// TwinCAT 3 PLC project PowerLink_v2
// ProgramVersion: 3.1.4023.0
// libraries:
//   EfficientIO Communicator, * (EfficientIO)
//   EfficientIO ModbusTCP, * (EfficientIO)
//   Lynus Persistent Data V1, * (Lynus AG)
//   Lynus Standards, * (EfficientIO)
//   Tc2_BABasic, * (Beckhoff Automation GmbH)
//   Tc2_ModbusSrv, * (Beckhoff Automation GmbH)
//   Tc2_Standard, * (Beckhoff Automation GmbH)
//   Tc2_System, * (Beckhoff Automation GmbH)
//   Tc2_Utilities, * (Beckhoff Automation GmbH)
//   Tc3_IotBase, * (Beckhoff Automation GmbH)
//   Tc3_IPCDiag, * (Beckhoff Automation GmbH)
//   Tc3_JsonXml, * (Beckhoff Automation GmbH)
//   Tc3_Module, * (Beckhoff Automation GmbH)
//   EfficientIO Energy Basic,1.0.0.4,EfficientIO
// project tree:
//   DUTs/ ST_Hoymiles_DTU_Pro_PV_OutData.TcDUT (not stored)
//   ENUMs/ E_State.TcDUT
//   ENUMs/Hoymiles/ E_Hoymiles_OperatingState.TcDUT, E_Hoymiles_PV_Error.TcDUT
//   / FastTask.TcTTO (not stored), MiddleTask.TcTTO (not stored), SlowTask.TcTTO (not stored)
//   FBs/ FB_Convert_Dword_Real.TcPOU, FB_EM24_DIN.TcPOU (not stored), FB_Enphase.TcPOU (not stored), FB_ECS_LIBREO.TcPOU, FB_Enphase_Helper.TcPOU (not stored), FB_ECS_LIBREO_Helper.TcPOU, FB_Hoymiles_DTU_ProS_PV_Inverter.TcPOU, FB_Hoymiles_DTU_ProS_PV_Inverter_inclWrite.TcPOU, FB_ModBus_100Registers_FC3_inclID.TcPOU (not stored), FB_PAC2200.TcPOU, prg_ReadDeviceName.TcPOU
//   POUs/ prgBattery.TcPOU (not stored), prgCalc.TcPOU, prgComEffIO.TcPOU, prgCS.TcPOU, prgEM.TcPOU, prgEMS.TcPOU, prgEnphase.TcPOU (not stored), prgPersistent.TcPOU, prgPV.TcPOU, prgRWEffIO.TcPOU (not stored), prgSystemTime.TcPOU (not stored), prgVarEffIO.TcPOU (not stored)

// ---- ENUMs/E_State.TcDUT
{attribute 'qualified_only'}
TYPE E_State :
(
	Init := 0,
	ReadOnce,
	Error,
	Idle,
	Wait

	
);
END_TYPE

// ---- ENUMs/Hoymiles/E_Hoymiles_OperatingState.TcDUT
{attribute 'qualified_only'}
{attribute 'strict'}
TYPE E_Hoymiles_OperatingState :
(
	eNoDataReceived := 0,
	eOff := 1,
	eSleeping := 2,
	eStartingUp := 3,
	eTrackingPowerPoint := 4,
	eForcedPowerReduction := 5,
	eShuttingDown := 6,
	eFaults := 7,
	eStandby := 8
);
END_TYPE

// ---- ENUMs/Hoymiles/E_Hoymiles_PV_Error.TcDUT
{attribute 'qualified_only'}
{attribute 'strict'}
TYPE E_Hoymiles_PV_Error :
(
	eNoError := 0,
	eModbusTCPError := 1,
	eHoymilesError := 2,
	eHoymilesTooBigValueReceived := 3
);
END_TYPE

// ---- FBs/FB_Convert_Dword_Real.TcPOU
FUNCTION_BLOCK FB_Convert_Dword_Real
VAR_INPUT
	word_In_1:	WORD;
	word_In_2:	WORD;
	e_ByteOrderIn	: eByteOrder;						//Byte Format
	
END_VAR
VAR_OUTPUT
	real_Output	:REAL;
END_VAR
VAR
	fbConvertWordToDword		: FB_CV_WORD_TO_DWORD;			//Convert Word to Dword
	usintSign					: USINT;						// converstion dword to real	
	intExponent					: INT;							// converstion dword to real
	realMantisse				: REAL;							// converstion dword to real
END_VAR

fbConvertWordToDword(wInputValue_1:= word_In_1, wInputValue_2:= word_In_2, eByteOrderForConvert:= e_ByteOrderIn , dwOutputValue=> );
(* Sign *)
usintSign:=BOOL_TO_USINT(fbConvertWordToDword.dwOutputValue.31);
(* Exponent *)
intExponent:=DWORD_TO_INT(SHR(fbConvertWordToDword.dwOutputValue,23) AND 16#FF);
(* Mantisse *)
realMantisse:=DWORD_TO_REAL(fbConvertWordToDword.dwOutputValue AND 16#7FFFFF);
(* Result *)
real_Output := LREAL_TO_REAL((EXPT((-1),usintSign) * (1+realMantisse/8388608) * EXPT(2,intExponent-127)));

END_FUNCTION_BLOCK

// ---- FBs/FB_ECS_LIBREO.TcPOU
FUNCTION_BLOCK FB_ECS_LIBREO
VAR_INPUT
	bStart				: BOOL;
	tDelayRequest		: TIME := T#1S;		//Timer for delay before start with the next read or write Request
	sHostname			: STRING(255);		//Hostname or IP Adress from the Server
END_VAR

VAR_IN_OUT
END_VAR

VAR_OUTPUT
	bValidResult				: BOOL;															//Valid Result received from Server
    bBusy						: BOOL;															//Function is Busy
    bError						: BOOL;															//Error sucess
	bDone						: BOOL;															//True after the decoding from the received Json File
	bConnected					: BOOL;															//Connection to the Server
	hrErrorCode       			: HRESULT;														//Error Result from Http Client
	
	bCarConnected				: BOOL;
	bCarCharging				: BOOL;
	lrTotalPower				: LREAL;
	uiChrgCurr					: UINT;
	uiExtChrgCurr				: UINT;
END_VAR

VAR
	fbClient					: FB_IotHttpClient;
	fbHttpGet					: FB_ECS_LIBREO_Helper;
	timStartRequest				: TON;															//Timer to Start the Request
	FPStartRequest				: R_TRIG;														//Internal positive Edge
	FPDone						: R_TRIG;														//Internal positive Edge
	FNStart						: F_TRIG;														//Internal negative Edge
END_VAR

(*------------------------------------------------------------------------------------Configure HTTP Client------------------------------------------------------------------------------------------------------*)

fbClient.sHostName := sHostname;
fbClient.tConnectionTimeout := tDelayRequest;

IF NOT fbClient.bConfigured THEN 
	fbClient.nHostPort:= 80;
	fbClient.bKeepAlive := TRUE;
	fbClient.tConnectionTimeout := T#2S;
END_IF


//Timer to start the Request
FPStartRequest(CLK:= bStart, Q=> );
	timStartRequest(IN:= fbClient.bConfigured AND bStart AND NOT timStartRequest.Q, PT:= tDelayRequest, Q=> , ET=> );
		IF ((timStartRequest.Q AND NOT bBusy) OR (FPStartRequest.Q AND NOT bBusy AND fbClient.bConfigured)) THEN fbHttpGet.bSend := TRUE; END_IF

				
//Http Get Function
fbHttpGet(
	bCarConnected => bCarConnected, 
	bCarCharging => bCarCharging,
	lrTotalPower => lrTotalPower,
	uiChrgCurr => uiChrgCurr,
	uiExtChrgCurr => uiExtChrgCurr,
	bSend:= , 
	fbClient:= fbClient, 
	bBusy=> bBusy, 
	bError=> ,
	sContent=> );

lrTotalPower := LIMIT( 0, lrTotalPower, lrTotalPower) / 1000;

fbHttpGet.bSend := FALSE;

FPDone(CLK:= bDone, Q=> );

fbClient.Execute();

//Error
IF fbHttpGet.bError OR fbClient.bError THEN bError := TRUE; ELSE bError := FALSE; END_IF	
	hrErrorCode := fbClient.hrErrorCode;

END_FUNCTION_BLOCK

// ---- FBs/FB_ECS_LIBREO_Helper.TcPOU
FUNCTION_BLOCK FB_ECS_LIBREO_Helper
VAR_INPUT
	bSend			: BOOL;
END_VAR

VAR_IN_OUT
	fbClient		: FB_IotHttpClient;
END_VAR

VAR_OUTPUT
	bBusy					: BOOL;
	bError					: BOOL;
	bCarConnected			: BOOL;
	bCarCharging			: BOOL;
	lrTotalPower			: LREAL;
	uiChrgCurr				: UINT;
	uiExtChrgCurr			: UINT;

END_VAR

VAR
	fbRequestStatus		: FB_IotHttpRequest;
	fbJson				: FB_JsonDomParser;
	nState				: UDINT;
	RisingEdge			: R_TRIG;
	timTimeout			: TON;
	tTimeOut			: TIME := T#30S;
	
	bGetContentResult	: BOOL;
	sContent			: STRING(2048);
	
	bGetJsonResult		: BOOL;
	jsonDoc				: SJsonValue;
	jsonVal				: SJsonValue;
	
	nReqCount			: UDINT;	
	nResCount			: UDINT;
	nValidResCount		: UDINT;
	nErrCount			: UDINT;
END_VAR

//Timer for Timeout
timTimeout(IN:= nState = 1 AND bBusy, PT:= tTimeOut, Q=> , ET=> );
	IF timTimeout.Q THEN 
		nState := 0;
		bBusy := FALSE;
	END_IF

RisingEdge(CLK:= bSend );
CASE nState OF
0:	
	IF RisingEdge.Q THEN 
		IF fbRequestStatus.SendRequest(sUri:='/status', fbClient:=fbClient, eRequestType:=ETcIotHttpRequestType.HTTP_Get, 0, 0, 0) THEN
			nState:= 1;
			nReqCount:= nReqCount+1;
			bBusy:= TRUE;
			bError:= FALSE;
		END_IF					
	END_IF
1:
	IF NOT fbRequestStatus.bBusy THEN
		bError:= TRUE;
		
		IF NOT fbRequestStatus.bError THEN				 
			bGetContentResult:= fbRequestStatus.GetContent(pContent:= ADR(sContent), nContentSize:= SIZEOF(sContent), bSetNullTermination:= TRUE);
			IF fbRequestStatus.nStatusCode >= 200 AND fbRequestStatus.nStatusCode < 300 THEN
				bGetJsonResult:= FALSE;
				jsonDoc:= fbRequestStatus.GetJsonDomContent(fbJson);
				IF jsonDoc <> 0 THEN
					bGetJsonResult:= TRUE;
					IF fbJson.HasMember(jsonDoc, 'ts')  THEN
						jsonVal:= fbJson.FindMember(jsonDoc, 'chrgCurr');
						nValidResCount:= nValidResCount+1;
						IF fbJson.IsUint(jsonVal) THEN							
							uiChrgCurr:= UDINT_TO_UINT(fbJson.GetUint(jsonVal));									
						END_IF
						jsonVal:= fbJson.FindMember(jsonDoc, 'extCurr');
						nValidResCount:= nValidResCount+1;
						IF fbJson.IsUint(jsonVal) THEN							
							uiExtChrgCurr:= UDINT_TO_UINT(fbJson.GetUint(jsonVal));									
						END_IF
						jsonVal:= fbJson.FindMember(jsonDoc, 'evConn');
						nValidResCount:= nValidResCount+1;
						IF fbJson.IsBool(jsonVal) THEN							
							bCarConnected:= fbJson.GetBool(jsonVal);									
						END_IF
						jsonVal:= fbJson.FindMember(jsonDoc, 'chrgState');
						nValidResCount:= nValidResCount+1;
						IF fbJson.IsBool(jsonVal) THEN							
							bCarCharging:= fbJson.GetBool(jsonVal);									
						END_IF
						jsonVal:= fbJson.FindMemberPath(jsonDoc, 'readings/wattTotal');
						nValidResCount:= nValidResCount+1;
						IF fbJson.IsDouble(jsonVal) THEN							
							lrTotalPower:= fbJson.GetDouble(jsonVal);									
						END_IF		
						bError:= FALSE;
					END_IF						
				nResCount:= nResCount+1;			
				END_IF
			END_IF
		END_IF
		
	nState:= 0;
	bBusy:= FALSE;
		IF bError THEN
			nErrCount:= nErrCount+1;
		END_IF
	END_IF  	
END_CASE

fbClient.Execute();

END_FUNCTION_BLOCK

// ---- FBs/FB_Hoymiles_DTU_ProS_PV_Inverter.TcPOU
FUNCTION_BLOCK FB_Hoymiles_DTU_ProS_PV_Inverter
VAR_INPUT PERSISTENT
	bEnable						: BOOL;												//True = Function is enabled, FALSE = Function is dissabled, no new Data
	sIPAdress					: STRING(15);										//IP Adress from the Inverter
	byUnitID_Inverter			: BYTE;												//Unit ID fromt the Inverter (1 to 247)
END_VAR
VAR_OUTPUT
	DataHoymiles_DTU_Pro_Total	: ST_Hoymiles_DTU_Pro_PV_OutData;					//Output structure with Data from Symo 10
	arrDataHoymiles_DTU_Pro		: ARRAY[1..30] OF ST_Hoymiles_DTU_Pro_PV_OutData;	//Output structure with Data 
	stDataEMPower_PV			: ST_ElectricMeter_Output_Power;					//Output structure with Data from Electric Meter PV (Power Data)
	stDataEMCounter_PV			: ST_ElectricMeter_Output_Counter;					//Output structure with Data from Electric Meter PV (Counter Data)
	diNrOfEM_OUT_PV				: DINT;												//Active Number from the Electric Meter for using on other functions
END_VAR
VAR
	fbElMeter					: FB_ElectricMeter;									//Electric Meter Function 
	fbNumberDevice				: FB_NumberOfDevice;								//Function block to calcualte the number of the Device
	fbConvertEnergyRegister		: FB_CV_WORD_TO_UDINT;								//Convert function
	fbMBRead_FC3				: FB_MBReadRegs;									//Modbus Read Function (FC3)
	timDelay					: TON;												//Timer for Delay between Requests
	timTimeout					: TON;												//Timer for Timeout
	timDissableFunctions		: TON;												//Timer to dissable the Function after Lynus_Standards.Constants_General.tTimeDissableLynusFunctions Days without connection to the Lynus Cloud
	timResetConnectionOnGVL		: TON;												//Timer to try reset the connection Flag on the GVL. (When somebody delete the Connection Function and make only a onlinechange)
	FPEnable					: R_TRIG;											//Internal positive Edge
	FPError_FC_3				: R_TRIG;											//Internal positive Edge
	PD_String					: FB_PersistentData_String;							//Function to save persistent data 
	arrBuffer_FC3				: ARRAY[1..100] OF WORD;							//Buffer with Data from FC3
	arrPD						: ARRAY[1..2] OF FB_PersistentData_Number;			//Function to save persistent data 
	byWaitInStep				: BYTE;												//Wait in Step before start to clean data on PLC
	iStateGVLData				: INT;												//State machine to handle the data on the GVL
	iStateModbus				: INT;												//State variable for Statemachine
	iStateModbus_CP				: INT;												//Compare State variable
	diCounterForGVL				: DINT;												//Counter to clean old data on GVL
	rValBefWToOut				: REAL;												//Value to check the received data from the inverter befor wirte to the output structure
	lrCheckValue				: LREAL;											//Internal Value to check the value before convert
	i: INT;
	timDelayError: TON;
	x: INT;

	timWait: Ton;
END_VAR

//Creator : Stefan Lackner
//Company : EfficientIO
//Date : 02.05.2023
//Version : 0.0.0.0  NOT TESTED

//With this function its possible to read out values from the Hoymiles DTU ProS Gateway
//The protocol to the Inverter is Modbus TCP
//Attention. To access the registers, an offset of 1 must always be subtracted. Register 40001 would then be on register 40000.

// operation state of the inverter is unclear if that is ok, no documentation from Hoymiles

//NOTE for diNr.....Designation => 
//_IN = Here Data come in from other Functions or go out to other functions about the GVL
//_OUT = Here Data go out to other functions about the GVL

(*------------------------------------------------------------------------------------------General Input Part---------------------------------------------------------------------------------------------*)

//Check limitation
byUnitID_Inverter := LIMIT(1,byUnitID_Inverter,254);

(*-------------------------------------------------------------Calcualte the number of EM System---------------------------------------------------------------*)

fbNumberDevice(
	diActualNumberOfDevices:= Lynus_Standards.GVL_Energy.stNumberOfDevices.diNumberOfElectricMeters, 
	diMaxNumberOfDevices:= Constants_Energy.diMaxNumberOfElectricMeters, 
	udiCounterOnlineChange:= TwinCAT_SystemInfoVarList._AppInfo.OnlineChangeCnt, 
	bNumberIsCalculatet=> , 
	bFPNumberIsCalculatet=> , 
	bOnlineChange=> , 
	diNumberForThisDevice=> diNrOfEM_OUT_PV, 
	diNumberOfTotalDevices=> );

//Write new Numer on GVL
IF fbNumberDevice.bFPNumberIsCalculatet THEN
	Lynus_Standards.GVL_Energy.stNumberOfDevices.diNumberOfElectricMeters := fbNumberDevice.diNumberOfTotalDevices;	
END_IF 

//Delete old Number on GVL
IF fbNumberDevice.bOnlineChange THEN 
	Lynus_Standards.GVL_Energy.stNumberOfDevices.diNumberOfElectricMeters := diNrOfEM_OUT_PV;	
	iStateGVLData := 1; 
END_IF

(*-------------------------------------------------------------Service from Backend is ready and check the connection to backen for dissabel/enable Function---------------------------------------------------------------*)

//Try to reset the variable for connection on the GVL. When all is normal then the Lynus Mqtt connection function set this variable to true in the next cycle
//When we have no connection to the backend then after Lynus_Standards.Constants_General.tTimeDissableLynusFunctions days the Function is dissabled with all of his functionalities
timResetConnectionOnGVL(IN:= NOT timResetConnectionOnGVL.Q, PT:= T#1H, Q=> , ET=> );
IF timResetConnectionOnGVL.Q THEN Lynus_Standards.GVL_Communicator.bStateConnectionToEnableFunctions := FALSE; END_IF
IF NOT Lynus_Standards.GVL_Communicator.bStateConnectionToEnableFunctions THEN timDissableFunctions.IN := TRUE; ELSE timDissableFunctions.IN := FALSE; END_IF  
timDissableFunctions(IN:= , PT:= Lynus_Standards.Constants_General.tTimeDissableLynusFunctions, Q=> , ET=> );
	
(*------------------------------------------------------------------------------------------State Machine---------------------------------------------------------------------------------------------*)
	
//Enable
FPEnable(CLK:= bEnable, Q=> );
IF FPEnable.Q AND iStateModbus = 0 THEN iStateModbus := 1; END_IF
IF NOT bEnable OR timDissableFunctions.Q THEN iStateModbus := 0; END_IF

//Timer for delay
timDelay(IN:= , PT:= T#100MS, Q=> , ET=> );	

//Timer for Timeout in Statemachine
IF iStateModbus = iStateModbus_CP THEN timTimeout.IN := TRUE; ELSE timTimeout.IN := FALSE; END_IF
IF iStateModbus = 0 THEN timTimeout.IN := FALSE; END_IF
timTimeout(IN:= , PT:= T#20S, Q=> , ET=> );	

//Timer for delay in error state
timDelayError(IN:= , PT:= T#1S, Q=> , ET=> );	

// Timer for wait between polls
timWait(In:= , PT:= T#1S, Q=>, ET=> );


//Statemachine
CASE iStateModbus OF
	
	0://Init Step
		iStateModbus_CP := iStateModbus;
		timDelay.IN := FALSE;
		
		DataHoymiles_DTU_Pro_Total.bFunctionIsActive := FALSE;
		DataHoymiles_DTU_Pro_Total.eOperatingState := E_Hoymiles_OperatingState.eNoDataReceived;
		fbMBRead_FC3.bExecute := FALSE;
		lrCheckValue := 0;
		rValBefWToOut := 0;
		
		// clean arrays
		FOR i:=1 TO 30 BY 1 DO
			arrDataHoymiles_DTU_Pro[i].bError := FALSE;
			arrDataHoymiles_DTU_Pro[i].bFunctionIsActive := FALSE;
			arrDataHoymiles_DTU_Pro[i].eErrorState := 0;
			arrDataHoymiles_DTU_Pro[i].eOperatingState := 0;
			arrDataHoymiles_DTU_Pro[i].iPortNumber := 0;
			arrDataHoymiles_DTU_Pro[i].lrGridFrequency := 0;
			arrDataHoymiles_DTU_Pro[i].lrGridVoltage := 0;			
			arrDataHoymiles_DTU_Pro[i].lrPowerAcInverter := 0;
			arrDataHoymiles_DTU_Pro[i].lrPVVoltage := 0;
			arrDataHoymiles_DTU_Pro[i].lrPVCurrent := 0;
		END_FOR
		timDelayError.IN := TRUE;
		IF timDelayError.Q THEN
			iStateModbus := 1;
			timDelayError.IN := FALSE;
		END_IF				
			
	1://Read out first Registers from 4096 
		DataHoymiles_DTU_Pro_Total.bFunctionIsActive := TRUE;
		iStateModbus_CP := iStateModbus;
		
		fbMBRead_FC3.nQuantity := 100;
		fbMBRead_FC3.nMBAddr := 4096;
		fbMBRead_FC3.bExecute := TRUE;
		fbMBRead_FC3.nUnitID := byUnitID_Inverter;
			
		IF fbMBRead_FC3.bBusy THEN timDelay.IN := TRUE; END_IF
		
		//Wait for Delay, copy Data and then next step
		IF NOT fbMBRead_FC3.bBusy AND NOT fbMBRead_FC3.bError AND timDelay.Q THEN 
			FOR i:= 0 TO 4 BY 1 DO		// 5 ports per poll
				// Port Number
				arrDataHoymiles_DTU_Pro[i+1].iPortNumber := BYTE_TO_INT( WORD_TO_BYTE(arrBuffer_FC3[4+20*i] AND 16#FFFF));
				IF arrDataHoymiles_DTU_Pro[i+1].iPortNumber  <>0 THEN
					//PV Voltage
					arrDataHoymiles_DTU_Pro[i+1].lrPVVoltage  := (WORD_TO_LREAL(arrBuffer_FC3[5+20*i]))/10;
					//PV Current
					arrDataHoymiles_DTU_Pro[i+1].lrPVCurrent := (WORD_TO_LREAL(arrBuffer_FC3[6+20*i]))/100;
					//Grid Voltage
					arrDataHoymiles_DTU_Pro[i+1].lrGridVoltage := (WORD_TO_LREAL(arrBuffer_FC3[7+20*i]))/10;
					//Grid Frequency
					arrDataHoymiles_DTU_Pro[i+1].lrGridFrequency  := (WORD_TO_LREAL(arrBuffer_FC3[8+20*i]))/100;
					//Copy Data AC Power
					arrDataHoymiles_DTU_Pro[i+1].lrPowerAcInverter := (WORD_TO_LREAL(arrBuffer_FC3[9+20*i]))/10000;
				
					//Copy Data AC production Energy
			//		fbConvertEnergyRegister(wInputValue_1:= arrBuffer_FC3[11+20*i], wInputValue_2:= arrBuffer_FC3[12+20*i], eByteOrderForConvert:= eByteOrder.eBigEndian, udiOutputValue=> );
			//		rValBefWToOut := UDINT_TO_REAL(fbConvertEnergyRegister.udiOutputValue);
			//		lrCheckValue := rValBefWToOut;	
			//		IF lrCheckValue >= - 3.402823E+38 AND lrCheckValue <= 3.402823E+38 THEN 
			//			arrDataHoymiles_DTU_Pro[i+1].lrPVProductionEnergy := lrCheckValue /1000 ;
						arrDataHoymiles_DTU_Pro[i+1].lrPVProductionEnergy := (WORD_TO_REAL(arrBuffer_FC3[11+20*i]) * 65536 + WORD_TO_REAL(arrBuffer_FC3[12+20*i])) /10; 
			//		ELSE
			//			arrDataHoymiles_DTU_Pro[i+6].eErrorState := E_Hoymiles_PV_Error.eHoymilesTooBigValueReceived;	
			//		END_IF
					
					
					//Operating State		--->>>>> needs to get checked with Hoymiles if the states are correct
					IF arrBuffer_FC3[14+20*i] = 1 THEN 
						arrDataHoymiles_DTU_Pro[i+1].eOperatingState := E_Hoymiles_OperatingState.eOff;
					ELSIF arrBuffer_FC3[14+20*i] = 2 THEN 
						arrDataHoymiles_DTU_Pro[i+1].eOperatingState := E_Hoymiles_OperatingState.eSleeping;
					ELSIF arrBuffer_FC3[14+20*i] = 3 THEN 
						arrDataHoymiles_DTU_Pro[i+1].eOperatingState := E_Hoymiles_OperatingState.eStartingUp;
					ELSIF arrBuffer_FC3[14+20*i] = 4 THEN 
						arrDataHoymiles_DTU_Pro[i+1].eOperatingState := E_Hoymiles_OperatingState.eTrackingPowerPoint;
					ELSIF arrBuffer_FC3[14+20*i] = 5 THEN 
						arrDataHoymiles_DTU_Pro[i+1].eOperatingState := E_Hoymiles_OperatingState.eForcedPowerReduction;
					ELSIF arrBuffer_FC3[14+20*i] = 6 THEN 
						arrDataHoymiles_DTU_Pro[i+1].eOperatingState := E_Hoymiles_OperatingState.eShuttingDown;
					ELSIF arrBuffer_FC3[14+20*i] = 7 THEN 
						arrDataHoymiles_DTU_Pro[i+1].eOperatingState := E_Hoymiles_OperatingState.eFaults;
					ELSIF arrBuffer_FC3[14+20*i] = 8 THEN 
						arrDataHoymiles_DTU_Pro[i+1].eOperatingState := E_Hoymiles_OperatingState.eStandby;
					ELSE 
						arrDataHoymiles_DTU_Pro[i+1].eOperatingState := E_Hoymiles_OperatingState.eNoDataReceived;
					END_IF
				ELSE
					arrDataHoymiles_DTU_Pro[i+1].lrPVVoltage := 0;
					arrDataHoymiles_DTU_Pro[i+1].lrPVCurrent := 0;
					arrDataHoymiles_DTU_Pro[i+1].lrGridVoltage := 0;
					arrDataHoymiles_DTU_Pro[i+1].lrGridFrequency  := 0;
					arrDataHoymiles_DTU_Pro[i+1].lrPowerAcInverter := 0;
					arrDataHoymiles_DTU_Pro[i+1].lrPVProductionEnergy := 0;
				END_IF
			END_FOR
			//Next Step
			IF iStateModbus = 1 THEN
				fbMBRead_FC3.bExecute := FALSE;
				timDelay.IN := FALSE;
				iStateModbus := 2;
				DataHoymiles_DTU_Pro_Total.bError := FALSE; 
				DataHoymiles_DTU_Pro_Total.eErrorState := E_Hoymiles_PV_Error.eNoError;
			END_IF
		END_IF
			

		//Error or Timeout
		IF FPError_FC_3.Q OR timTimeout.Q THEN
			iStateModbus := 300;
			DataHoymiles_DTU_Pro_Total.eErrorState := E_Hoymiles_PV_Error.eModbusTCPError;
		END_IF

	2://Wait and back to 1 step or next ports poll
		iStateModbus_CP := iStateModbus;
		timWait.IN := TRUE;
		IF arrBuffer_FC3[82] <> 0 AND timWait.Q THEN // if the last port hast a serial number, so to the next 5 ports needs to get checked 
			timWait.IN := FALSE;
			iStateModbus := 3;
		ELSIF timWait.Q  THEN
			timWait.IN := FALSE;
			iStateModbus := 1;
		END_IF
	
	3://Read out second 100 Registers from 4296 
		DataHoymiles_DTU_Pro_Total.bFunctionIsActive := TRUE;
		iStateModbus_CP := iStateModbus;
		
		fbMBRead_FC3.nQuantity := 100;
		fbMBRead_FC3.nMBAddr := 4296;
		fbMBRead_FC3.bExecute := TRUE;
		fbMBRead_FC3.nUnitID := byUnitID_Inverter;
			
		IF fbMBRead_FC3.bBusy THEN timDelay.IN := TRUE; END_IF
		
		//Wait for Delay, copy Data and then next step
		IF NOT fbMBRead_FC3.bBusy AND NOT fbMBRead_FC3.bError AND timDelay.Q THEN 
			FOR i:= 0 TO 4 BY 1 DO		// 5 ports per poll
				// Port Number
				arrDataHoymiles_DTU_Pro[i+6].iPortNumber := BYTE_TO_INT( WORD_TO_BYTE(arrBuffer_FC3[4+20*i] AND 16#FFFF));
				IF arrDataHoymiles_DTU_Pro[i+6].iPortNumber <>0 THEN
					//PV Voltage
					arrDataHoymiles_DTU_Pro[i+6].lrPVVoltage  := (WORD_TO_LREAL(arrBuffer_FC3[5+20*i]))/10;
					//PV Current
					arrDataHoymiles_DTU_Pro[i+6].lrPVCurrent := (WORD_TO_LREAL(arrBuffer_FC3[6+20*i]))/100;
					//Grid Voltage
					arrDataHoymiles_DTU_Pro[i+6].lrGridVoltage := (WORD_TO_LREAL(arrBuffer_FC3[7+20*i]))/10;
					//Grid Frequency
					arrDataHoymiles_DTU_Pro[i+6].lrGridFrequency  := (WORD_TO_LREAL(arrBuffer_FC3[8+20*i]))/100;
					//Copy Data AC Power
					arrDataHoymiles_DTU_Pro[i+6].lrPowerAcInverter := (WORD_TO_LREAL(arrBuffer_FC3[9+20*i]))/10000;
				
					//Copy Data AC production Energy
			//		fbConvertEnergyRegister(wInputValue_1:= arrBuffer_FC3[11+20*i], wInputValue_2:= arrBuffer_FC3[12+20*i], eByteOrderForConvert:= eByteOrder.eBigEndian, udiOutputValue=> );
			//		rValBefWToOut := UDINT_TO_REAL(fbConvertEnergyRegister.udiOutputValue);
			//		lrCheckValue := rValBefWToOut;	
			//		IF lrCheckValue >= - 3.402823E+38 AND lrCheckValue <= 3.402823E+38 THEN 
			//			arrDataHoymiles_DTU_Pro[i+6].lrPVProductionEnergy := lrCheckValue /1000 ;
						arrDataHoymiles_DTU_Pro[i+6].lrPVProductionEnergy := (WORD_TO_REAL(arrBuffer_FC3[11+20*i]) * 65536 + WORD_TO_REAL(arrBuffer_FC3[12+20*i])) /10; 
			//		ELSE
			//			arrDataHoymiles_DTU_Pro[i+6].eErrorState := E_Hoymiles_PV_Error.eHoymilesTooBigValueReceived;	
			//		END_IF
					
					
					//Operating State		--->>>>> needs to get checked with Hoymiles if the states are correct
					IF arrBuffer_FC3[14+20*i] = 1 THEN 
						arrDataHoymiles_DTU_Pro[i+6].eOperatingState := E_Hoymiles_OperatingState.eOff;
					ELSIF arrBuffer_FC3[14+20*i] = 2 THEN 
						arrDataHoymiles_DTU_Pro[i+6].eOperatingState := E_Hoymiles_OperatingState.eSleeping;
					ELSIF arrBuffer_FC3[14+20*i] = 3 THEN 
						arrDataHoymiles_DTU_Pro[i+6].eOperatingState := E_Hoymiles_OperatingState.eStartingUp;
					ELSIF arrBuffer_FC3[14+20*i] = 4 THEN 
						arrDataHoymiles_DTU_Pro[i+6].eOperatingState := E_Hoymiles_OperatingState.eTrackingPowerPoint;
					ELSIF arrBuffer_FC3[14+20*i] = 5 THEN 
						arrDataHoymiles_DTU_Pro[i+6].eOperatingState := E_Hoymiles_OperatingState.eForcedPowerReduction;
					ELSIF arrBuffer_FC3[14+20*i] = 6 THEN 
						arrDataHoymiles_DTU_Pro[i+6].eOperatingState := E_Hoymiles_OperatingState.eShuttingDown;
					ELSIF arrBuffer_FC3[14+20*i] = 7 THEN 
						arrDataHoymiles_DTU_Pro[i+6].eOperatingState := E_Hoymiles_OperatingState.eFaults;
					ELSIF arrBuffer_FC3[14+20*i] = 8 THEN 
						arrDataHoymiles_DTU_Pro[i+6].eOperatingState := E_Hoymiles_OperatingState.eStandby;
					ELSE 
						arrDataHoymiles_DTU_Pro[i+6].eOperatingState := E_Hoymiles_OperatingState.eNoDataReceived;
					END_IF
				ELSE
					arrDataHoymiles_DTU_Pro[i+6].lrPVVoltage := 0;
					arrDataHoymiles_DTU_Pro[i+6].lrPVCurrent := 0;
					arrDataHoymiles_DTU_Pro[i+6].lrGridVoltage := 0;
					arrDataHoymiles_DTU_Pro[i+6].lrGridFrequency  := 0;
					arrDataHoymiles_DTU_Pro[i+6].lrPowerAcInverter := 0;
					arrDataHoymiles_DTU_Pro[i+6].lrPVProductionEnergy := 0;
				END_IF
			END_FOR
			//Next Step
			IF iStateModbus = 3 THEN
				fbMBRead_FC3.bExecute := FALSE;
				timDelay.IN := FALSE;
				iStateModbus := 4;
				DataHoymiles_DTU_Pro_Total.bError := FALSE; 
				DataHoymiles_DTU_Pro_Total.eErrorState := E_Hoymiles_PV_Error.eNoError;
			END_IF
		END_IF
		//Error or Timeout
		IF FPError_FC_3.Q OR timTimeout.Q THEN
			iStateModbus := 300;
			DataHoymiles_DTU_Pro_Total.eErrorState := E_Hoymiles_PV_Error.eModbusTCPError;
		END_IF
		
	4://Wait and back to 1 step
		iStateModbus_CP := iStateModbus;
		timWait.IN := TRUE;
		IF  arrBuffer_FC3[82] <> 0 AND timWait.Q THEN // if the last port hast a serial number, bo to the next 5 ports 
			timWait.IN := FALSE;
			iStateModbus := 1;		// change to state 5 and add the polls accordingly
		ELSIF timWait.Q  THEN
			timWait.IN := FALSE;
			iStateModbus := 1;
		END_IF
				
	300://Error
		iStateModbus_CP := iStateModbus;
		timDelay.IN := FALSE;
		fbMBRead_FC3.bExecute := FALSE;
		DataHoymiles_DTU_Pro_Total.bError := TRUE;
		timDelayError.IN := TRUE;
		IF timDelayError.Q THEN
			iStateModbus := 0;
			timDelayError.IN := FALSE;
		END_IF
							
END_CASE

(*------------------------------------------------------------------------------------------Modbus TCP Function---------------------------------------------------------------------------------------------*)

fbMBRead_FC3(	sIPAddr:= sIPAdress, 
				nTCPPort:= 502, 
				cbLength:= SIZEOF(arrBuffer_FC3), 
				pDestAddr:= ADR(arrBuffer_FC3), 
				tTimeout:= T#10S );
				
FPError_FC_3(CLK:= fbMBRead_FC3.bError, Q=> );

(*----------------------------------------------------------------------------------------Electric Meter Data----------------------------------------------------------------------------------------------*)

//Error and Warning
IF timDissableFunctions.Q THEN fbElMeter.bWarning := TRUE; fbElMeter.iWarningCode := 0; ELSE fbElMeter.bWarning := FALSE; END_IF   
IF DataHoymiles_DTU_Pro_Total.bError OR Lynus_Standards.GVL_Energy.stNumberOfDevices.diNumberOfElectricMeters > Constants_Energy.diMaxNumberOfElectricMeters THEN fbElMeter.bError := TRUE; ELSE fbElMeter.bError := FALSE; END_IF  

IF Lynus_Standards.GVL_Energy.stNumberOfDevices.diNumberOfElectricMeters > Constants_Energy.diMaxNumberOfElectricMeters THEN 
	fbElMeter.iErrorCode := 1;
ELSIF DataHoymiles_DTU_Pro_Total.bError THEN 
	fbElMeter.iErrorCode := 0;
END_IF  

//Read Out Data done for EM Function
IF iStateModbus <> 2 THEN fbElMeter.bReadOutDataDone := TRUE; ELSE fbElMeter.bReadOutDataDone := FALSE; END_IF

//Function block for meter data
IF iStateModbus = 2 OR iStateModbus = 4 THEN 
	fbElMeter.lrPowerTotal := 0;
	fbElMeter.lrFrequency := 0;
	FOR i:= 1 TO 30 BY 1 DO
		fbElMeter.lrPowerTotal := arrDataHoymiles_DTU_Pro[i].lrPowerAcInverter + fbElMeter.lrPowerTotal;
		IF arrDataHoymiles_DTU_Pro[i].lrGridFrequency > 45 AND arrDataHoymiles_DTU_Pro[i].lrGridFrequency < 55 THEN
			fbElMeter.lrFrequency := arrDataHoymiles_DTU_Pro[i].lrGridFrequency;
		END_IF
		IF arrDataHoymiles_DTU_Pro[i].lrGridVoltage >150 AND arrDataHoymiles_DTU_Pro[i].lrGridVoltage < 300 THEN
			fbElMeter.lrVoltageL1N := arrDataHoymiles_DTU_Pro[i].lrGridVoltage;
		END_IF
	END_FOR
END_IF
	
fbElMeter(
	bEnable:= bEnable AND NOT timDissableFunctions.Q, 
	bError:= , 
	bEnableReadOutFunction:= FALSE, 
	bWriteWithDelay:= TRUE,
	bPowerDataInvers:= TRUE, 
	bReadOutDataDone:= ,
	iTimeReadOutInterval:= , 
	iErrorCode:= , 
	iWarningCode:= , 
	lrTotalCounterEnergy_Consumption:= 0, 
	lrTotalCounterEnergy_Production:= , 
	lrCounterEnergyT1_Consumption:= 0, 
	lrCounterEnergyT2_Consumption:= 0, 
	lrCounterEnergyT1_Production:= , 
	lrCounterEnergyT2_Production:= 0, 
	lrCurrentL1:= 0, 
	lrVoltageL1N:= , 
	lrVoltageL1L2:= 0, 
	lrPowerL1:= 0, 
	lrCurrentL2:= 0, 
	lrVoltageL2N:= 0 , 
	lrVoltageL2L3:= 0 , 
	lrPowerL2:= 0, 
	lrCurrentL3:= 0 , 
	lrVoltageL3N:= 0, 
	lrVoltageL3L1:= 0, 
	lrPowerL3:= 0, 
	lrPowerTotal:= , 
	lrFrequency:= , 
	lrReactivePowerTotal:= 0, 
	lrApparentPowerTotal:= 0, 
	tTimDelayOutput:= T#5S, 
	stDataEMOutPower=> , 
	stDataEMOutPowerDelay=> stDataEMPower_PV, 
	stDataEMOutCounter=> ,
	stDataEMOutCounterDelay=> stDataEMCounter_PV, 
	bReadOutMeter=> );
DataHoymiles_DTU_Pro_Total.lrGridFrequency 		:= fbElMeter.lrFrequency;
DataHoymiles_DTU_Pro_Total.lrGridVoltage		:= fbElMeter.lrVoltageL1N;
DataHoymiles_DTU_Pro_Total.lrPowerAcInverter	:= fbElMeter.lrPowerTotal;
DataHoymiles_DTU_Pro_Total.lrPVProductionEnergy := stDataEMCounter_PV.lrTotalCounterEnergy_Production;

(*-----------------------------------------------------------Handle data to Global structure for the Electric Meter system-----------------------------------------------------------------*)

CASE iStateGVLData OF
	
	0://Init Step
		byWaitInStep := 0;
		diCounterForGVL := 1;
	
	1://Wait for 4 Steps before clean al Data on GVL
		byWaitInStep := byWaitInStep + 1;
		IF byWaitInStep >= 4 AND fbNumberDevice.bNumberIsCalculatet THEN iStateGVLData := 2; END_IF
		//To much Devices, back to the Init step
		IF byWaitInStep >= 4 AND NOT fbNumberDevice.bNumberIsCalculatet THEN iStateGVLData := 0; END_IF	
		
	2://Clear all Data in GVL
		Lynus_Standards.GVL_Energy.stDataElectricMeters[diCounterForGVL].bEnabled := FALSE;	
		Lynus_Standards.GVL_Energy.stDataElectricMeters[diCounterForGVL].byErrorWarning := 0;
		Lynus_Standards.GVL_Energy.stDataElectricMeters[diCounterForGVL].lrCounterEnergyT1_Consumption := 0;
		Lynus_Standards.GVL_Energy.stDataElectricMeters[diCounterForGVL].lrCounterEnergyT1_Production := 0;
		Lynus_Standards.GVL_Energy.stDataElectricMeters[diCounterForGVL].lrCounterEnergyT2_Consumption := 0;
		Lynus_Standards.GVL_Energy.stDataElectricMeters[diCounterForGVL].lrCounterEnergyT2_Production := 0;
		Lynus_Standards.GVL_Energy.stDataElectricMeters[diCounterForGVL].lrPower := 0;
		Lynus_Standards.GVL_Energy.stDataElectricMeters[diCounterForGVL].lrPowerConsumption := 0;
		Lynus_Standards.GVL_Energy.stDataElectricMeters[diCounterForGVL].lrPowerConsumption := 0;
		Lynus_Standards.GVL_Energy.stDataElectricMeters[diCounterForGVL].lrPowerProduction := 0;
		Lynus_Standards.GVL_Energy.stDataElectricMeters[diCounterForGVL].lrTotalCounterEnergy_Consumption := 0;
		Lynus_Standards.GVL_Energy.stDataElectricMeters[diCounterForGVL].lrTotalCounterEnergy_Production := 0;
		
		diCounterForGVL := diCounterForGVL + 1;
		diCounterForGVL := LIMIT(0,diCounterForGVL,Constants_Energy.diMaxNumberOfElectricMeters);
		//Back to the init step
		IF diCounterForGVL >= Constants_Energy.diMaxNumberOfElectricMeters THEN iStateGVLData := 0; END_IF
		
END_CASE 	 

IF diNrOfEM_OUT_PV > 0 AND fbNumberDevice.bNumberIsCalculatet THEN
	Lynus_Standards.GVL_Energy.stDataElectricMeters[diNrOfEM_OUT_PV].bEnabled := fbElMeter.stDataEMOutPower.bEnabled;
	Lynus_Standards.GVL_Energy.stDataElectricMeters[diNrOfEM_OUT_PV].byErrorWarning := fbElMeter.stDataEMOutPower.byErrorWarning;
	Lynus_Standards.GVL_Energy.stDataElectricMeters[diNrOfEM_OUT_PV].lrCounterEnergyT1_Consumption := fbElMeter.stDataEMOutCounter.lrCounterEnergyT1_Consumption;
	Lynus_Standards.GVL_Energy.stDataElectricMeters[diNrOfEM_OUT_PV].lrCounterEnergyT1_Production := fbElMeter.stDataEMOutCounter.lrCounterEnergyT1_Production;
	Lynus_Standards.GVL_Energy.stDataElectricMeters[diNrOfEM_OUT_PV].lrCounterEnergyT2_Consumption := fbElMeter.stDataEMOutCounter.lrCounterEnergyT2_Consumption;
	Lynus_Standards.GVL_Energy.stDataElectricMeters[diNrOfEM_OUT_PV].lrCounterEnergyT2_Production := fbElMeter.stDataEMOutCounter.lrCounterEnergyT2_Production;		
	Lynus_Standards.GVL_Energy.stDataElectricMeters[diNrOfEM_OUT_PV].lrPower := fbElMeter.stDataEMOutPower.lrPowerTotal;
	Lynus_Standards.GVL_Energy.stDataElectricMeters[diNrOfEM_OUT_PV].lrPowerConsumption := fbElMeter.stDataEMOutPower.lrPowerConsumption;
	Lynus_Standards.GVL_Energy.stDataElectricMeters[diNrOfEM_OUT_PV].lrPowerProduction := fbElMeter.stDataEMOutPower.lrPowerProduction;
	Lynus_Standards.GVL_Energy.stDataElectricMeters[diNrOfEM_OUT_PV].lrTotalCounterEnergy_Consumption := fbElMeter.stDataEMOutCounter.lrTotalCounterEnergy_Consumption;
	Lynus_Standards.GVL_Energy.stDataElectricMeters[diNrOfEM_OUT_PV].lrTotalCounterEnergy_Production := fbElMeter.stDataEMOutCounter.lrTotalCounterEnergy_Production;
END_IF

(*----------------------------------------------------------Save persistent data----------------------------------------------------------------*)

arrPD[1](lrValue:= BOOL_TO_LREAL(bEnable), bEventBasedActive=> );
arrPD[2](lrValue:= BYTE_TO_LREAL(byUnitID_Inverter), bEventBasedActive=> );
PD_String(sText:= sIPAdress, bEventBasedActive=> );

END_FUNCTION_BLOCK

// ---- FBs/FB_Hoymiles_DTU_ProS_PV_Inverter_inclWrite.TcPOU
FUNCTION_BLOCK FB_Hoymiles_DTU_ProS_PV_Inverter_inclWrite
VAR_INPUT PERSISTENT
	bEnable						: BOOL;												//True = Function is enabled, FALSE = Function is dissabled, no new Data
	sIPAdress					: STRING(15);										//IP Adress from the Inverter
	byUnitID_Inverter			: BYTE;												//Unit ID fromt the Inverter (1 to 247)
	byte_Setpoint				: BYTE;
END_VAR
VAR_OUTPUT
	DataHoymiles_DTU_Pro_Total	: ST_Hoymiles_DTU_Pro_PV_OutData;					//Output structure with Data from Symo 10
	arrDataHoymiles_DTU_Pro		: ARRAY[1..30] OF ST_Hoymiles_DTU_Pro_PV_OutData;	//Output structure with Data 
	stDataEMPower_PV			: ST_ElectricMeter_Output_Power;					//Output structure with Data from Electric Meter PV (Power Data)
	stDataEMCounter_PV			: ST_ElectricMeter_Output_Counter;					//Output structure with Data from Electric Meter PV (Counter Data)
	diNrOfEM_OUT_PV				: DINT;												//Active Number from the Electric Meter for using on other functions
END_VAR
VAR
	fbElMeter					: FB_ElectricMeter;									//Electric Meter Function 
	fbNumberDevice				: FB_NumberOfDevice;								//Function block to calcualte the number of the Device
	fbConvertEnergyRegister		: FB_CV_WORD_TO_UDINT;								//Convert function
	fbMBRead_FC3				: FB_MBReadRegs;									//Modbus Read Function (FC3)
	timDelay					: TON;												//Timer for Delay between Requests
	timTimeout					: TON;												//Timer for Timeout
	timDissableFunctions		: TON;												//Timer to dissable the Function after Lynus_Standards.Constants_General.tTimeDissableLynusFunctions Days without connection to the Lynus Cloud
	timResetConnectionOnGVL		: TON;												//Timer to try reset the connection Flag on the GVL. (When somebody delete the Connection Function and make only a onlinechange)
	FPEnable					: R_TRIG;											//Internal positive Edge
	FPError_FC_3				: R_TRIG;											//Internal positive Edge
	FPError_FC_6				: R_TRIG;											//Internal positive Edge
	PD_String					: FB_PersistentData_String;							//Function to save persistent data 
	arrBuffer_FC3				: ARRAY[1..100] OF WORD;							//Buffer with Data from FC3
	arrPD						: ARRAY[1..2] OF FB_PersistentData_Number;			//Function to save persistent data 
	byWaitInStep				: BYTE;												//Wait in Step before start to clean data on PLC
	iStateGVLData				: INT;												//State machine to handle the data on the GVL
	iStateModbus				: INT;												//State variable for Statemachine
	iStateModbus_CP				: INT;												//Compare State variable
	iStateModbusWrite			: INT;												//State variable for Statemachine
	diCounterForGVL				: DINT;												//Counter to clean old data on GVL
	rValBefWToOut				: REAL;												//Value to check the received data from the inverter befor wirte to the output structure
	lrCheckValue				: LREAL;											//Internal Value to check the value before convert
	i: INT;
	timDelayError: TON;
	x: INT;
	int_WriteSucessCounter: INT;
	fbMBWrite_FC6				: FB_MBWriteSingleReg;									//Modbus Write Function (FC16)
	timWait: Ton;
	
	wordBuffer_FC6				: WORD;								//Buffer with Data from FC6
	ton_Wait_write: Ton;
	tonDelayWrite: Ton;
	int_Error_Counter_Write: INT;
	ton_Wait_AfterWrite: TON;
END_VAR

//Creator : Stefan Lackner
//Company : EfficientIO
//Date : 02.05.2023
//Version : 0.0.0.0  NOT TESTED

//With this function its possible to read out values from the Hoymiles DTU ProS Gateway
//The protocol to the Inverter is Modbus TCP
//Attention. To access the registers, an offset of 1 must always be subtracted. Register 40001 would then be on register 40000.

// operation state of the inverter is unclear if that is ok, no documentation from Hoymiles

//NOTE for diNr.....Designation => 
//_IN = Here Data come in from other Functions or go out to other functions about the GVL
//_OUT = Here Data go out to other functions about the GVL

(*------------------------------------------------------------------------------------------General Input Part---------------------------------------------------------------------------------------------*)

//Check limitation
byUnitID_Inverter := LIMIT(1,byUnitID_Inverter,254);

(*-------------------------------------------------------------Calcualte the number of EM System---------------------------------------------------------------*)

fbNumberDevice(
	diActualNumberOfDevices:= Lynus_Standards.GVL_Energy.stNumberOfDevices.diNumberOfElectricMeters, 
	diMaxNumberOfDevices:= Constants_Energy.diMaxNumberOfElectricMeters, 
	udiCounterOnlineChange:= TwinCAT_SystemInfoVarList._AppInfo.OnlineChangeCnt, 
	bNumberIsCalculatet=> , 
	bFPNumberIsCalculatet=> , 
	bOnlineChange=> , 
	diNumberForThisDevice=> diNrOfEM_OUT_PV, 
	diNumberOfTotalDevices=> );

//Write new Numer on GVL
IF fbNumberDevice.bFPNumberIsCalculatet THEN
	Lynus_Standards.GVL_Energy.stNumberOfDevices.diNumberOfElectricMeters := fbNumberDevice.diNumberOfTotalDevices;	
END_IF 

//Delete old Number on GVL
IF fbNumberDevice.bOnlineChange THEN 
	Lynus_Standards.GVL_Energy.stNumberOfDevices.diNumberOfElectricMeters := diNrOfEM_OUT_PV;	
	iStateGVLData := 1; 
END_IF

(*-------------------------------------------------------------Service from Backend is ready and check the connection to backen for dissabel/enable Function---------------------------------------------------------------*)

//Try to reset the variable for connection on the GVL. When all is normal then the Lynus Mqtt connection function set this variable to true in the next cycle
//When we have no connection to the backend then after Lynus_Standards.Constants_General.tTimeDissableLynusFunctions days the Function is dissabled with all of his functionalities
timResetConnectionOnGVL(IN:= NOT timResetConnectionOnGVL.Q, PT:= T#1H, Q=> , ET=> );
IF timResetConnectionOnGVL.Q THEN Lynus_Standards.GVL_Communicator.bStateConnectionToEnableFunctions := FALSE; END_IF
IF NOT Lynus_Standards.GVL_Communicator.bStateConnectionToEnableFunctions THEN timDissableFunctions.IN := TRUE; ELSE timDissableFunctions.IN := FALSE; END_IF  
timDissableFunctions(IN:= , PT:= Lynus_Standards.Constants_General.tTimeDissableLynusFunctions, Q=> , ET=> );
	
(*------------------------------------------------------------------------------------------State Machine---------------------------------------------------------------------------------------------*)
	
//Enable
FPEnable(CLK:= bEnable, Q=> );
IF FPEnable.Q AND iStateModbus = 0 THEN iStateModbus := 1; END_IF
IF NOT bEnable OR timDissableFunctions.Q THEN iStateModbus := 0; END_IF

//Timer for delay
timDelay(IN:= , PT:= T#100MS, Q=> , ET=> );	
tonDelayWrite(IN:= , PT:= T#100MS, Q=> , ET=> );	

//Timer for Timeout in Statemachine
IF iStateModbus = iStateModbus_CP THEN timTimeout.IN := TRUE; ELSE timTimeout.IN := FALSE; END_IF
IF iStateModbus = 0 THEN timTimeout.IN := FALSE; END_IF
timTimeout(IN:= , PT:= T#20S, Q=> , ET=> );	

//Timer for delay in error state
timDelayError(IN:= , PT:= T#1S, Q=> , ET=> );	

// Timer for wait between polls
timWait(In:= , PT:= T#1S, Q=>, ET=> );


//Statemachine
CASE iStateModbus OF
	
	0://Init Step
		iStateModbus_CP := iStateModbus;
		timDelay.IN := FALSE;
		
		DataHoymiles_DTU_Pro_Total.bFunctionIsActive := FALSE;
		DataHoymiles_DTU_Pro_Total.eOperatingState := E_Hoymiles_OperatingState.eNoDataReceived;
		fbMBRead_FC3.bExecute := FALSE;
		lrCheckValue := 0;
		rValBefWToOut := 0;
		
		// clean arrays
		FOR i:=1 TO 30 BY 1 DO
			arrDataHoymiles_DTU_Pro[i].bError := FALSE;
			arrDataHoymiles_DTU_Pro[i].bFunctionIsActive := FALSE;
			arrDataHoymiles_DTU_Pro[i].eErrorState := 0;
			arrDataHoymiles_DTU_Pro[i].eOperatingState := 0;
			arrDataHoymiles_DTU_Pro[i].iPortNumber := 0;
			arrDataHoymiles_DTU_Pro[i].lrGridFrequency := 0;
			arrDataHoymiles_DTU_Pro[i].lrGridVoltage := 0;			
			arrDataHoymiles_DTU_Pro[i].lrPowerAcInverter := 0;
			arrDataHoymiles_DTU_Pro[i].lrPVVoltage := 0;
			arrDataHoymiles_DTU_Pro[i].lrPVCurrent := 0;
		END_FOR
		timDelayError.IN := TRUE;
		IF timDelayError.Q THEN
			iStateModbus := 1;
			timDelayError.IN := FALSE;
		END_IF				
			
	1://Read out first Registers from 4096 
		DataHoymiles_DTU_Pro_Total.bFunctionIsActive := TRUE;
		iStateModbus_CP := iStateModbus;
		
		fbMBRead_FC3.nQuantity := 100;
		fbMBRead_FC3.nMBAddr := 4096;
		fbMBRead_FC3.bExecute := TRUE;
		fbMBRead_FC3.nUnitID := byUnitID_Inverter;
			
		IF fbMBRead_FC3.bBusy THEN timDelay.IN := TRUE; END_IF
		
		//Wait for Delay, copy Data and then next step
		IF NOT fbMBRead_FC3.bBusy AND NOT fbMBRead_FC3.bError AND timDelay.Q THEN 
			FOR i:= 0 TO 4 BY 1 DO		// 5 ports per poll
				// Port Number
				arrDataHoymiles_DTU_Pro[i+1].iPortNumber := BYTE_TO_INT( WORD_TO_BYTE(arrBuffer_FC3[4+20*i] AND 16#FFFF));
				IF arrDataHoymiles_DTU_Pro[i+1].iPortNumber  <>0 THEN
					//PV Voltage
					arrDataHoymiles_DTU_Pro[i+1].lrPVVoltage  := (WORD_TO_LREAL(arrBuffer_FC3[5+20*i]))/10;
					//PV Current
					arrDataHoymiles_DTU_Pro[i+1].lrPVCurrent := (WORD_TO_LREAL(arrBuffer_FC3[6+20*i]))/100;
					//Grid Voltage
					arrDataHoymiles_DTU_Pro[i+1].lrGridVoltage := (WORD_TO_LREAL(arrBuffer_FC3[7+20*i]))/10;
					//Grid Frequency
					arrDataHoymiles_DTU_Pro[i+1].lrGridFrequency  := (WORD_TO_LREAL(arrBuffer_FC3[8+20*i]))/100;
					//Copy Data AC Power
					arrDataHoymiles_DTU_Pro[i+1].lrPowerAcInverter := (WORD_TO_LREAL(arrBuffer_FC3[9+20*i]))/10000;
				
					//Copy Data AC production Energy
			//		fbConvertEnergyRegister(wInputValue_1:= arrBuffer_FC3[11+20*i], wInputValue_2:= arrBuffer_FC3[12+20*i], eByteOrderForConvert:= eByteOrder.eBigEndian, udiOutputValue=> );
			//		rValBefWToOut := UDINT_TO_REAL(fbConvertEnergyRegister.udiOutputValue);
			//		lrCheckValue := rValBefWToOut;	
			//		IF lrCheckValue >= - 3.402823E+38 AND lrCheckValue <= 3.402823E+38 THEN 
			//			arrDataHoymiles_DTU_Pro[i+1].lrPVProductionEnergy := lrCheckValue /1000 ;
						arrDataHoymiles_DTU_Pro[i+1].lrPVProductionEnergy := (WORD_TO_REAL(arrBuffer_FC3[11+20*i]) * 65536 + WORD_TO_REAL(arrBuffer_FC3[12+20*i])) /10; 
			//		ELSE
			//			arrDataHoymiles_DTU_Pro[i+6].eErrorState := E_Hoymiles_PV_Error.eHoymilesTooBigValueReceived;	
			//		END_IF
					
					
					//Operating State		--->>>>> needs to get checked with Hoymiles if the states are correct
					IF arrBuffer_FC3[14+20*i] = 1 THEN 
						arrDataHoymiles_DTU_Pro[i+1].eOperatingState := E_Hoymiles_OperatingState.eOff;
					ELSIF arrBuffer_FC3[14+20*i] = 2 THEN 
						arrDataHoymiles_DTU_Pro[i+1].eOperatingState := E_Hoymiles_OperatingState.eSleeping;
					ELSIF arrBuffer_FC3[14+20*i] = 3 THEN 
						arrDataHoymiles_DTU_Pro[i+1].eOperatingState := E_Hoymiles_OperatingState.eStartingUp;
					ELSIF arrBuffer_FC3[14+20*i] = 4 THEN 
						arrDataHoymiles_DTU_Pro[i+1].eOperatingState := E_Hoymiles_OperatingState.eTrackingPowerPoint;
					ELSIF arrBuffer_FC3[14+20*i] = 5 THEN 
						arrDataHoymiles_DTU_Pro[i+1].eOperatingState := E_Hoymiles_OperatingState.eForcedPowerReduction;
					ELSIF arrBuffer_FC3[14+20*i] = 6 THEN 
						arrDataHoymiles_DTU_Pro[i+1].eOperatingState := E_Hoymiles_OperatingState.eShuttingDown;
					ELSIF arrBuffer_FC3[14+20*i] = 7 THEN 
						arrDataHoymiles_DTU_Pro[i+1].eOperatingState := E_Hoymiles_OperatingState.eFaults;
					ELSIF arrBuffer_FC3[14+20*i] = 8 THEN 
						arrDataHoymiles_DTU_Pro[i+1].eOperatingState := E_Hoymiles_OperatingState.eStandby;
					ELSE 
						arrDataHoymiles_DTU_Pro[i+1].eOperatingState := E_Hoymiles_OperatingState.eNoDataReceived;
					END_IF
				ELSE
					arrDataHoymiles_DTU_Pro[i+1].lrPVVoltage := 0;
					arrDataHoymiles_DTU_Pro[i+1].lrPVCurrent := 0;
					arrDataHoymiles_DTU_Pro[i+1].lrGridVoltage := 0;
					arrDataHoymiles_DTU_Pro[i+1].lrGridFrequency  := 0;
					arrDataHoymiles_DTU_Pro[i+1].lrPowerAcInverter := 0;
					arrDataHoymiles_DTU_Pro[i+1].lrPVProductionEnergy := 0;
				END_IF
			END_FOR
			//Next Step
			IF iStateModbus = 1 THEN
				fbMBRead_FC3.bExecute := FALSE;
				timDelay.IN := FALSE;
				iStateModbus := 2;
				DataHoymiles_DTU_Pro_Total.bError := FALSE; 
				DataHoymiles_DTU_Pro_Total.eErrorState := E_Hoymiles_PV_Error.eNoError;
			END_IF
		END_IF
			

		//Error or Timeout
		IF FPError_FC_3.Q OR timTimeout.Q THEN
			iStateModbus := 300;
			DataHoymiles_DTU_Pro_Total.eErrorState := E_Hoymiles_PV_Error.eModbusTCPError;
		END_IF

	2://Wait and back to 1 step or next ports poll
		iStateModbus_CP := iStateModbus;
		timWait.IN := TRUE;
		IF arrBuffer_FC3[82] <> 0 AND timWait.Q THEN // if the last port hast a serial number, so to the next 5 ports needs to get checked 
			timWait.IN := FALSE;
			iStateModbus := 3;
		ELSIF timWait.Q  THEN
			timWait.IN := FALSE;
			iStateModbusWrite := 1;
			iStateModbus := -1;
			iStateModbus_CP := iStateModbus;
			// iStateModbus := 1;
		END_IF
	
	3://Read out second 100 Registers from 4296 
		DataHoymiles_DTU_Pro_Total.bFunctionIsActive := TRUE;
		iStateModbus_CP := iStateModbus;
		
		fbMBRead_FC3.nQuantity := 100;
		fbMBRead_FC3.nMBAddr := 4296;
		fbMBRead_FC3.bExecute := TRUE;
		fbMBRead_FC3.nUnitID := byUnitID_Inverter;
			
		IF fbMBRead_FC3.bBusy THEN timDelay.IN := TRUE; END_IF
		
		//Wait for Delay, copy Data and then next step
		IF NOT fbMBRead_FC3.bBusy AND NOT fbMBRead_FC3.bError AND timDelay.Q THEN 
			FOR i:= 0 TO 4 BY 1 DO		// 5 ports per poll
				// Port Number
				arrDataHoymiles_DTU_Pro[i+6].iPortNumber := BYTE_TO_INT( WORD_TO_BYTE(arrBuffer_FC3[4+20*i] AND 16#FFFF));
				IF arrDataHoymiles_DTU_Pro[i+6].iPortNumber <>0 THEN
					//PV Voltage
					arrDataHoymiles_DTU_Pro[i+6].lrPVVoltage  := (WORD_TO_LREAL(arrBuffer_FC3[5+20*i]))/10;
					//PV Current
					arrDataHoymiles_DTU_Pro[i+6].lrPVCurrent := (WORD_TO_LREAL(arrBuffer_FC3[6+20*i]))/100;
					//Grid Voltage
					arrDataHoymiles_DTU_Pro[i+6].lrGridVoltage := (WORD_TO_LREAL(arrBuffer_FC3[7+20*i]))/10;
					//Grid Frequency
					arrDataHoymiles_DTU_Pro[i+6].lrGridFrequency  := (WORD_TO_LREAL(arrBuffer_FC3[8+20*i]))/100;
					//Copy Data AC Power
					arrDataHoymiles_DTU_Pro[i+6].lrPowerAcInverter := (WORD_TO_LREAL(arrBuffer_FC3[9+20*i]))/10000;
				
					//Copy Data AC production Energy
			//		fbConvertEnergyRegister(wInputValue_1:= arrBuffer_FC3[11+20*i], wInputValue_2:= arrBuffer_FC3[12+20*i], eByteOrderForConvert:= eByteOrder.eBigEndian, udiOutputValue=> );
			//		rValBefWToOut := UDINT_TO_REAL(fbConvertEnergyRegister.udiOutputValue);
			//		lrCheckValue := rValBefWToOut;	
			//		IF lrCheckValue >= - 3.402823E+38 AND lrCheckValue <= 3.402823E+38 THEN 
			//			arrDataHoymiles_DTU_Pro[i+6].lrPVProductionEnergy := lrCheckValue /1000 ;
						arrDataHoymiles_DTU_Pro[i+6].lrPVProductionEnergy := (WORD_TO_REAL(arrBuffer_FC3[11+20*i]) * 65536 + WORD_TO_REAL(arrBuffer_FC3[12+20*i])) /10; 
			//		ELSE
			//			arrDataHoymiles_DTU_Pro[i+6].eErrorState := E_Hoymiles_PV_Error.eHoymilesTooBigValueReceived;	
			//		END_IF
					
					
					//Operating State		--->>>>> needs to get checked with Hoymiles if the states are correct
					IF arrBuffer_FC3[14+20*i] = 1 THEN 
						arrDataHoymiles_DTU_Pro[i+6].eOperatingState := E_Hoymiles_OperatingState.eOff;
					ELSIF arrBuffer_FC3[14+20*i] = 2 THEN 
						arrDataHoymiles_DTU_Pro[i+6].eOperatingState := E_Hoymiles_OperatingState.eSleeping;
					ELSIF arrBuffer_FC3[14+20*i] = 3 THEN 
						arrDataHoymiles_DTU_Pro[i+6].eOperatingState := E_Hoymiles_OperatingState.eStartingUp;
					ELSIF arrBuffer_FC3[14+20*i] = 4 THEN 
						arrDataHoymiles_DTU_Pro[i+6].eOperatingState := E_Hoymiles_OperatingState.eTrackingPowerPoint;
					ELSIF arrBuffer_FC3[14+20*i] = 5 THEN 
						arrDataHoymiles_DTU_Pro[i+6].eOperatingState := E_Hoymiles_OperatingState.eForcedPowerReduction;
					ELSIF arrBuffer_FC3[14+20*i] = 6 THEN 
						arrDataHoymiles_DTU_Pro[i+6].eOperatingState := E_Hoymiles_OperatingState.eShuttingDown;
					ELSIF arrBuffer_FC3[14+20*i] = 7 THEN 
						arrDataHoymiles_DTU_Pro[i+6].eOperatingState := E_Hoymiles_OperatingState.eFaults;
					ELSIF arrBuffer_FC3[14+20*i] = 8 THEN 
						arrDataHoymiles_DTU_Pro[i+6].eOperatingState := E_Hoymiles_OperatingState.eStandby;
					ELSE 
						arrDataHoymiles_DTU_Pro[i+6].eOperatingState := E_Hoymiles_OperatingState.eNoDataReceived;
					END_IF
				ELSE
					arrDataHoymiles_DTU_Pro[i+6].lrPVVoltage := 0;
					arrDataHoymiles_DTU_Pro[i+6].lrPVCurrent := 0;
					arrDataHoymiles_DTU_Pro[i+6].lrGridVoltage := 0;
					arrDataHoymiles_DTU_Pro[i+6].lrGridFrequency  := 0;
					arrDataHoymiles_DTU_Pro[i+6].lrPowerAcInverter := 0;
					arrDataHoymiles_DTU_Pro[i+6].lrPVProductionEnergy := 0;
				END_IF
			END_FOR
			//Next Step
			IF iStateModbus = 3 THEN
				fbMBRead_FC3.bExecute := FALSE;
				timDelay.IN := FALSE;
				iStateModbus := 4;
				DataHoymiles_DTU_Pro_Total.bError := FALSE; 
				DataHoymiles_DTU_Pro_Total.eErrorState := E_Hoymiles_PV_Error.eNoError;
			END_IF
		END_IF
		//Error or Timeout
		IF FPError_FC_3.Q OR timTimeout.Q THEN
			iStateModbus := 300;
			DataHoymiles_DTU_Pro_Total.eErrorState := E_Hoymiles_PV_Error.eModbusTCPError;
		END_IF
		
	4://Wait and back to 1 step
		iStateModbus_CP := iStateModbus;
		timWait.IN := TRUE;
		IF  arrBuffer_FC3[82] <> 0 AND timWait.Q THEN // if the last port hast a serial number, bo to the next 5 ports 
			timWait.IN := FALSE;
			iStateModbus := 1;		// change to state 5 and add the polls accordingly
		ELSIF timWait.Q  THEN
			timWait.IN := FALSE;
			iStateModbus := -1;
			iStateModbusWrite := 1;
			iStateModbus_CP := iStateModbus;
		//	iStateModbus := 1;
		END_IF
				
	300://Error
		iStateModbus_CP := iStateModbus;
		timDelay.IN := FALSE;
		fbMBRead_FC3.bExecute := FALSE;
		DataHoymiles_DTU_Pro_Total.bError := TRUE;
		timDelayError.IN := TRUE;
		IF timDelayError.Q THEN
			iStateModbus := 0;
			timDelayError.IN := FALSE;
		END_IF
							
END_CASE

(*------------------------------------------------------------------------------------------WriteFunction---------------------------------------------------------------------------------------------*)

	
CASE iStateModbusWrite OF	
	1://Search the Unit ID to read out the Data for each Inverter with Unit ID <> 0
		//iStateModbus_CP := iStateModbusWrite;
		byte_Setpoint := LIMIT (0,byte_Setpoint,100);
		
		iStateModbusWrite := 2;
				

	2://write setpoint
		//iStateModbus_CP := iStateModbusWrite;	

		wordBuffer_FC6 := BYTE_TO_WORD(byte_Setpoint);


		fbMBWrite_FC6.nMBAddr := 16#C001;
		fbMBWrite_FC6.bExecute := TRUE;
		fbMBWrite_FC6.nValue:= wordBuffer_FC6; 

				
		IF fbMBWrite_FC6.bBusy THEN 
			tonDelayWrite.IN := TRUE; 
		END_IF
	
		//Wait for Delay and then next step
		IF NOT fbMBWrite_FC6.bBusy AND NOT fbMBWrite_FC6.bError AND tonDelayWrite.Q THEN

			int_WriteSucessCounter :=int_WriteSucessCounter+1;
			
			fbMBWrite_FC6.bExecute := FALSE;
			tonDelayWrite.IN := FALSE;
			//Restart from new with the Read out part
			iStateModbusWrite := 3;
		END_IF
				
		//Error or Timout
		IF FPError_FC_6.Q OR timTimeout.Q THEN
			fbMBWrite_FC6.bExecute := FALSE;
			tonDelayWrite.IN := FALSE;
			iStateModbusWrite := 300;
		END_IF
	
	3:
		ton_Wait_AfterWrite.IN:=TRUE;
		IF ton_Wait_AfterWrite.Q THEN
			ton_Wait_AfterWrite.IN:=FALSE;
			iStateModbus := 1;
			iStateModbusWrite := 0;
		END_IF
		
		
	300:   // error
		int_Error_Counter_Write := int_Error_Counter_Write+1;
		iStateModbus := 1;
		iStateModbusWrite := 0;
END_CASE
ton_Wait_AfterWrite(pt:= T#2S);


(*------------------------------------------------------------------------------------------Modbus TCP Function---------------------------------------------------------------------------------------------*)

fbMBRead_FC3(	sIPAddr:= sIPAdress, 
				nTCPPort:= 502, 
				cbLength:= SIZEOF(arrBuffer_FC3), 
				pDestAddr:= ADR(arrBuffer_FC3), 
				tTimeout:= T#10S );
				
FPError_FC_3(CLK:= fbMBRead_FC3.bError, Q=> );

fbMBWrite_FC6(
	sIPAddr:= sIPAdress , 
	nTCPPort:= 502, 
	nUnitID:= byUnitID_Inverter, 
	nMBAddr:= , 
	nValue:= , 
	bExecute:= , 
	tTimeout:= T#5S, 
	bBusy=> , 
	bError=> , 
	nErrId=> );


		
FPError_FC_6(CLK:= fbMBWrite_FC6.bError, Q=> );



(*----------------------------------------------------------------------------------------Electric Meter Data----------------------------------------------------------------------------------------------*)

//Error and Warning
IF timDissableFunctions.Q THEN fbElMeter.bWarning := TRUE; fbElMeter.iWarningCode := 0; ELSE fbElMeter.bWarning := FALSE; END_IF   
IF DataHoymiles_DTU_Pro_Total.bError OR Lynus_Standards.GVL_Energy.stNumberOfDevices.diNumberOfElectricMeters > Constants_Energy.diMaxNumberOfElectricMeters THEN fbElMeter.bError := TRUE; ELSE fbElMeter.bError := FALSE; END_IF  

IF Lynus_Standards.GVL_Energy.stNumberOfDevices.diNumberOfElectricMeters > Constants_Energy.diMaxNumberOfElectricMeters THEN 
	fbElMeter.iErrorCode := 1;
ELSIF DataHoymiles_DTU_Pro_Total.bError THEN 
	fbElMeter.iErrorCode := 0;
END_IF  

//Read Out Data done for EM Function
IF iStateModbus <> 2 THEN fbElMeter.bReadOutDataDone := TRUE; ELSE fbElMeter.bReadOutDataDone := FALSE; END_IF

//Function block for meter data
IF iStateModbus = 2 OR iStateModbus = 4 THEN 
	fbElMeter.lrPowerTotal := 0;
	fbElMeter.lrFrequency := 0;
	FOR i:= 1 TO 30 BY 1 DO
		fbElMeter.lrPowerTotal := arrDataHoymiles_DTU_Pro[i].lrPowerAcInverter + fbElMeter.lrPowerTotal;
		IF arrDataHoymiles_DTU_Pro[i].lrGridFrequency > 45 AND arrDataHoymiles_DTU_Pro[i].lrGridFrequency < 55 THEN
			fbElMeter.lrFrequency := arrDataHoymiles_DTU_Pro[i].lrGridFrequency;
		END_IF
		IF arrDataHoymiles_DTU_Pro[i].lrGridVoltage >150 AND arrDataHoymiles_DTU_Pro[i].lrGridVoltage < 300 THEN
			fbElMeter.lrVoltageL1N := arrDataHoymiles_DTU_Pro[i].lrGridVoltage;
		END_IF
	END_FOR
END_IF
	
fbElMeter(
	bEnable:= bEnable AND NOT timDissableFunctions.Q, 
	bError:= , 
	bEnableReadOutFunction:= FALSE, 
	bWriteWithDelay:= TRUE,
	bPowerDataInvers:= TRUE, 
	bReadOutDataDone:= ,
	iTimeReadOutInterval:= , 
	iErrorCode:= , 
	iWarningCode:= , 
	lrTotalCounterEnergy_Consumption:= 0, 
	lrTotalCounterEnergy_Production:= , 
	lrCounterEnergyT1_Consumption:= 0, 
	lrCounterEnergyT2_Consumption:= 0, 
	lrCounterEnergyT1_Production:= , 
	lrCounterEnergyT2_Production:= 0, 
	lrCurrentL1:= 0, 
	lrVoltageL1N:= , 
	lrVoltageL1L2:= 0, 
	lrPowerL1:= 0, 
	lrCurrentL2:= 0, 
	lrVoltageL2N:= 0 , 
	lrVoltageL2L3:= 0 , 
	lrPowerL2:= 0, 
	lrCurrentL3:= 0 , 
	lrVoltageL3N:= 0, 
	lrVoltageL3L1:= 0, 
	lrPowerL3:= 0, 
	lrPowerTotal:= , 
	lrFrequency:= , 
	lrReactivePowerTotal:= 0, 
	lrApparentPowerTotal:= 0, 
	tTimDelayOutput:= T#5S, 
	stDataEMOutPower=> , 
	stDataEMOutPowerDelay=> stDataEMPower_PV, 
	stDataEMOutCounter=> ,
	stDataEMOutCounterDelay=> stDataEMCounter_PV, 
	bReadOutMeter=> );
DataHoymiles_DTU_Pro_Total.lrGridFrequency 		:= fbElMeter.lrFrequency;
DataHoymiles_DTU_Pro_Total.lrGridVoltage		:= fbElMeter.lrVoltageL1N;
DataHoymiles_DTU_Pro_Total.lrPowerAcInverter	:= fbElMeter.lrPowerTotal;
DataHoymiles_DTU_Pro_Total.lrPVProductionEnergy := stDataEMCounter_PV.lrTotalCounterEnergy_Production;

(*-----------------------------------------------------------Handle data to Global structure for the Electric Meter system-----------------------------------------------------------------*)

CASE iStateGVLData OF
	
	0://Init Step
		byWaitInStep := 0;
		diCounterForGVL := 1;
	
	1://Wait for 4 Steps before clean al Data on GVL
		byWaitInStep := byWaitInStep + 1;
		IF byWaitInStep >= 4 AND fbNumberDevice.bNumberIsCalculatet THEN iStateGVLData := 2; END_IF
		//To much Devices, back to the Init step
		IF byWaitInStep >= 4 AND NOT fbNumberDevice.bNumberIsCalculatet THEN iStateGVLData := 0; END_IF	
		
	2://Clear all Data in GVL
		Lynus_Standards.GVL_Energy.stDataElectricMeters[diCounterForGVL].bEnabled := FALSE;	
		Lynus_Standards.GVL_Energy.stDataElectricMeters[diCounterForGVL].byErrorWarning := 0;
		Lynus_Standards.GVL_Energy.stDataElectricMeters[diCounterForGVL].lrCounterEnergyT1_Consumption := 0;
		Lynus_Standards.GVL_Energy.stDataElectricMeters[diCounterForGVL].lrCounterEnergyT1_Production := 0;
		Lynus_Standards.GVL_Energy.stDataElectricMeters[diCounterForGVL].lrCounterEnergyT2_Consumption := 0;
		Lynus_Standards.GVL_Energy.stDataElectricMeters[diCounterForGVL].lrCounterEnergyT2_Production := 0;
		Lynus_Standards.GVL_Energy.stDataElectricMeters[diCounterForGVL].lrPower := 0;
		Lynus_Standards.GVL_Energy.stDataElectricMeters[diCounterForGVL].lrPowerConsumption := 0;
		Lynus_Standards.GVL_Energy.stDataElectricMeters[diCounterForGVL].lrPowerConsumption := 0;
		Lynus_Standards.GVL_Energy.stDataElectricMeters[diCounterForGVL].lrPowerProduction := 0;
		Lynus_Standards.GVL_Energy.stDataElectricMeters[diCounterForGVL].lrTotalCounterEnergy_Consumption := 0;
		Lynus_Standards.GVL_Energy.stDataElectricMeters[diCounterForGVL].lrTotalCounterEnergy_Production := 0;
		
		diCounterForGVL := diCounterForGVL + 1;
		diCounterForGVL := LIMIT(0,diCounterForGVL,Constants_Energy.diMaxNumberOfElectricMeters);
		//Back to the init step
		IF diCounterForGVL >= Constants_Energy.diMaxNumberOfElectricMeters THEN iStateGVLData := 0; END_IF
		
END_CASE 	 

IF diNrOfEM_OUT_PV > 0 AND fbNumberDevice.bNumberIsCalculatet THEN
	Lynus_Standards.GVL_Energy.stDataElectricMeters[diNrOfEM_OUT_PV].bEnabled := fbElMeter.stDataEMOutPower.bEnabled;
	Lynus_Standards.GVL_Energy.stDataElectricMeters[diNrOfEM_OUT_PV].byErrorWarning := fbElMeter.stDataEMOutPower.byErrorWarning;
	Lynus_Standards.GVL_Energy.stDataElectricMeters[diNrOfEM_OUT_PV].lrCounterEnergyT1_Consumption := fbElMeter.stDataEMOutCounter.lrCounterEnergyT1_Consumption;
	Lynus_Standards.GVL_Energy.stDataElectricMeters[diNrOfEM_OUT_PV].lrCounterEnergyT1_Production := fbElMeter.stDataEMOutCounter.lrCounterEnergyT1_Production;
	Lynus_Standards.GVL_Energy.stDataElectricMeters[diNrOfEM_OUT_PV].lrCounterEnergyT2_Consumption := fbElMeter.stDataEMOutCounter.lrCounterEnergyT2_Consumption;
	Lynus_Standards.GVL_Energy.stDataElectricMeters[diNrOfEM_OUT_PV].lrCounterEnergyT2_Production := fbElMeter.stDataEMOutCounter.lrCounterEnergyT2_Production;		
	Lynus_Standards.GVL_Energy.stDataElectricMeters[diNrOfEM_OUT_PV].lrPower := fbElMeter.stDataEMOutPower.lrPowerTotal;
	Lynus_Standards.GVL_Energy.stDataElectricMeters[diNrOfEM_OUT_PV].lrPowerConsumption := fbElMeter.stDataEMOutPower.lrPowerConsumption;
	Lynus_Standards.GVL_Energy.stDataElectricMeters[diNrOfEM_OUT_PV].lrPowerProduction := fbElMeter.stDataEMOutPower.lrPowerProduction;
	Lynus_Standards.GVL_Energy.stDataElectricMeters[diNrOfEM_OUT_PV].lrTotalCounterEnergy_Consumption := fbElMeter.stDataEMOutCounter.lrTotalCounterEnergy_Consumption;
	Lynus_Standards.GVL_Energy.stDataElectricMeters[diNrOfEM_OUT_PV].lrTotalCounterEnergy_Production := fbElMeter.stDataEMOutCounter.lrTotalCounterEnergy_Production;
END_IF

(*----------------------------------------------------------Save persistent data----------------------------------------------------------------*)

arrPD[1](lrValue:= BOOL_TO_LREAL(bEnable), bEventBasedActive=> );
arrPD[2](lrValue:= BYTE_TO_LREAL(byUnitID_Inverter), bEventBasedActive=> );
PD_String(sText:= sIPAdress, bEventBasedActive=> );

END_FUNCTION_BLOCK

// ---- FBs/FB_PAC2200.TcPOU
FUNCTION_BLOCK FB_PAC2200
VAR_INPUT PERSISTENT
	m_Enable					: BOOL;						//Enable the Fuctionblock and his logic
	str_IPAdress				: STRING(15);				//IP Adress of the meter
END_VAR
VAR_OUTPUT
	real_RealPower_kW				: REAL;					// Real power in W
	real_RealPowerL1_kW				: REAL;					// Real power in W
	real_RealPowerL2_kW				: REAL;					// Real power in W
	real_RealPowerL3_kW				: REAL;					// Real power in W
	real_ReactivePower_kVAr			: REAL;					// Reactive power in VAr
	real_ApparentPower_kVA			: REAL;					// Apparent power in VA
	real_Frequency_Hz				: REAL;					// Frequency in Hz
	real_VoltageL1N_V				: REAL;					//  Voltage L1-N in V 
	real_VoltageL2N_V				: REAL;					//  Voltage L2-N in V 
	real_VoltageL3N_V				: REAL;					//  Voltage L3-N in V 
	real_VoltageL1L2_V				: REAL;					//  Voltage L1-L2 in V 
	real_VoltageL2L3_V				: REAL;					//  Voltage L2-L3 in V 
	real_VoltageL3L1_V				: REAL;					//  Voltage L3-L1 in V 
	real_CurrentL1_A				: REAL;					//  Current L1 in A
	real_CurrentL2_A				: REAL;					//  Current L2 in A
	real_CurrentL3_A				: REAL;					//  Current L3 in A
	real_EnergyTotal_Import_T1_kWh	: REAL;					// Energy total in Wh
	real_EnergyTotal_Import_T2_kWh	: REAL;					// Energy total in Wh
	real_EnergyTotal_Export_T1_kWh	: REAL;					// Energy total in Wh
	real_EnergyTotal_Export_T2_kWh	: REAL;					// Energy total in Wh
	
	m_PollSuccessful				: BOOL;					// Poll succesfull		
	udint_Error_ID					: UDINT;				// ERR ID FB_MBReadRegs
END_VAR
VAR
//	{attribute 'hide'}
	w_Adress					: WORD;						//modbus adress
//	{attribute 'hide'}
	usint_Quantity				: USINT;					//Number of Words to get polled, max 100
//	{attribute 'hide'}
	fb_Convert_Data				: FB_Convert_Dword_Real;
//	{attribute 'hide'}
	e_ByteOrderConvert	: eByteOrder;						//Byte Format
//	{attribute 'hide'}
	timer_Delay					: TON;						//Timer for Delay between Requests
//	{attribute 'hide'}
	timer_DelayStart			: TON;						//Timer to start the state machine with Delay after enabling or after the system ist restartet
//	{attribute 'hide'}
	timer_TimeOut				: TON;						//Timer for Timeout MB Read
//	{attribute 'hide'}
	iStateModbusRead			: INT;						//State machine for read out Data over Modbus RTU
//	{attribute 'hide'}
	fbMBRead_FC3				: FB_MBReadRegs  ;		//Modbus Read Function (FC3)
//	{attribute 'hide'}
	ftrig_PEnable				: f_trig;					//Internal positive Edge
//	{attribute 'hide'}
	iStateModbusError			: INT;						//State machine for error out Data over Modbus TCP/IP	
//	{attribute 'hide'}
	FPError_FC_3				: R_TRIG;					//Internal positive Edge
//	{attribute 'hide'}
	arrBuffer_FC3				: ARRAY[0..100] OF WORD;		//Buffer with Data from FC3
//	{attribute 'hide'}
	arrBuffer_Received			: ARRAY[1..2,0..100] OF WORD;		//Total received Data
//	{attribute 'hide'}
	timer_Connection_ok			: TON;
//	{attribute 'hide'}
	int_Data_Received			: INT;
//	{attribute 'hide'}
	m_MBTCPError				: BOOL;
//	{attribute 'hide'}
	int_Data_Received_old		: INT;
//	{attribute 'hide'}
	timer_Connection_ok_TOF	: TOF;
//	{attribute 'hide'}
	m_Poll_ok: BOOL;
//	{attribute 'hide'}
	timer_Wait: Ton;
//	{attribute 'hide'}
	int_TimeoutError: INT;
//	{attribute 'hide'}
	int_FC4Error: INT;
//	{attribute 'hide'}
	i: INT;
//	{attribute 'hide'}
	x: INT;

END_VAR

// v0.1 by Stefan Lackner 20230714
// untested
// reads out Siemens PC2200 Multimeters


(*--------------------------------------------------------------------------------------------Limits-------------------------------------------------------------------------------------*)
w_Adress := LIMIT(0,w_Adress,65000);
usint_Quantity := LIMIT(1,usint_Quantity,100);
	
(*--------------------------------------------------------------------------------------------State Machine Read--------------------------------------------------------------------------------------*)

//Timer for Delay
timer_Delay(IN:= , PT:= T#50MS, Q=> , ET=> );

//Timeout Timer is dissabled when the Init Step is aktiv or the function is not enabled
IF iStateModbusRead = 0 OR NOT m_Enable THEN 
	timer_Timeout.IN := FALSE; 
END_IF
timer_Timeout(IN:= , PT:= T#1S, Q=> , ET=> );

//Enable with Delay that not all sockets have to be created at the same time
timer_DelayStart(IN:= m_Enable, PT:= T#1S, Q=> , ET=> );
ftrig_PEnable(CLK:= timer_DelayStart.Q, Q=> );

IF ftrig_PEnable.Q AND iStateModbusRead = 0 THEN 
	iStateModbusRead := 1; 
END_IF		
		
//Not Enabled
IF NOT m_Enable THEN 
	iStateModbusRead := 0; 
	iStateModbusError := 0; 
END_IF		
		
CASE iStateModbusRead OF

	0://Init Step 
		timer_Delay.IN := FALSE;
		fbMBRead_FC3.bExecute := FALSE;
		m_Poll_ok:=FALSE;
		int_Data_Received:=0;
		iStateModbusRead := iStateModbusRead+1;

	1: // clean the array  Poll 1
		FOR i:=0 TO 100 BY 1 DO
			arrBuffer_FC3[i] := 0;
		END_FOR
		w_Adress := 1;
		usint_Quantity := 100; 
		iStateModbusRead := iStateModbusRead+1;
		
	2://read the required registers
		//Start Read Poll 1
		fbMBRead_FC3.nQuantity := usint_Quantity;
		fbMBRead_FC3.nMBAddr := w_Adress;
		fbMBRead_FC3.bExecute := TRUE;
		fbMBRead_FC3.nUnitID := 1;
		timer_Timeout.IN := TRUE;
		IF fbMBRead_FC3.bBusy THEN 
			timer_Delay.IN := TRUE; 
		END_IF
		
		//Wait for Delay, copy Data and then next step
		IF NOT fbMBRead_FC3.bBusy AND NOT fbMBRead_FC3.bError AND timer_Delay.Q THEN
			m_Poll_ok:=TRUE;
			int_Data_Received:=int_Data_Received+1;
			m_MBTCPError := FALSE; 
			
			FOR i:=0 TO 100 BY 1 DO
				arrBuffer_Received[1,i] := arrBuffer_FC3[i];
			END_FOR
			
			//Go to Next Step
			timer_Timeout.IN := FALSE;
			fbMBRead_FC3.bExecute := FALSE;
			timer_Delay.IN := FALSE;		
			iStateModbusRead := iStateModbusRead+1;
		END_IF	

		//Error or Timeout
		IF FPError_FC_3.Q THEN 
			iStateModbusError := 300;
			int_FC4Error := int_FC4Error+1;
		ELSIF timer_Timeout.Q THEN  
			timer_Timeout.IN := FALSE; 	
			iStateModbusError := 300;
			int_TimeoutError := int_TimeoutError+1;
		END_IF
	
	3://Wait and go to next step
		timer_Wait.IN := TRUE;
		
		IF timer_Wait.Q = TRUE THEN
			iStateModbusRead := iStateModbusRead+1;
			timer_Wait.IN :=FALSE;
		END_IF

	4: // clean the array  Poll 2
		FOR i:=0 TO 100 BY 1 DO
			arrBuffer_FC3[i] := 0;
		END_FOR
		w_Adress := 2801;;
		usint_Quantity := 10; 
		iStateModbusRead := iStateModbusRead+1;
		
	5://read the required registers
		//Start Read Poll 2
		fbMBRead_FC3.nQuantity := usint_Quantity;
		fbMBRead_FC3.nMBAddr := w_Adress;
		fbMBRead_FC3.bExecute := TRUE;
		fbMBRead_FC3.nUnitID := 1;
		timer_Timeout.IN := TRUE;
		IF fbMBRead_FC3.bBusy THEN 
			timer_Delay.IN := TRUE; 
		END_IF
		
		//Wait for Delay, copy Data and then next step
		IF NOT fbMBRead_FC3.bBusy AND NOT fbMBRead_FC3.bError AND timer_Delay.Q THEN
			m_Poll_ok:=TRUE;
			int_Data_Received:=int_Data_Received+1;
			m_MBTCPError := FALSE; 
			
			FOR i:=0 TO 9 BY 1 DO
				arrBuffer_Received[2,i] := arrBuffer_FC3[i];
			END_FOR
			
			//Go to Next Step
			timer_Timeout.IN := FALSE;
			fbMBRead_FC3.bExecute := FALSE;
			timer_Delay.IN := FALSE;		
			iStateModbusRead := iStateModbusRead+1;
		END_IF	

		//Error or Timeout
		IF FPError_FC_3.Q THEN 
			iStateModbusError := 300;
			int_FC4Error := int_FC4Error+1;
		ELSIF timer_Timeout.Q THEN  
			timer_Timeout.IN := FALSE; 	
			iStateModbusError := 300;
			int_TimeoutError := int_TimeoutError+1;
		END_IF
	
	6://Wait and go to next step
		timer_Wait.IN := TRUE;
		
		IF timer_Wait.Q = TRUE THEN
			iStateModbusRead := 30;
			timer_Wait.IN :=FALSE;
		END_IF
		

	
	30: // convert data
		e_ByteOrderConvert := 0;
		x:=0;
		fb_Convert_Data(	word_In_1:= arrBuffer_Received[1,x], 
							word_In_2:= arrBuffer_Received[1,x+1], 
							e_ByteOrderIn:= e_ByteOrderConvert, 
							real_Output=> real_VoltageL1N_V);
		x:=x+2;
		fb_Convert_Data(	word_In_1:= arrBuffer_Received[1,x], 
							word_In_2:= arrBuffer_Received[1,x+1], 
							e_ByteOrderIn:= e_ByteOrderConvert, 
							real_Output=> real_VoltageL2N_V);
		x:=x+2;
		fb_Convert_Data(	word_In_1:= arrBuffer_Received[1,x], 
							word_In_2:= arrBuffer_Received[1,x+1], 
							e_ByteOrderIn:= e_ByteOrderConvert, 
							real_Output=> real_VoltageL3N_V);		
		x:=x+2;
		fb_Convert_Data(	word_In_1:= arrBuffer_Received[1,x], 
							word_In_2:= arrBuffer_Received[1,x+1], 
							e_ByteOrderIn:= e_ByteOrderConvert, 
							real_Output=> real_VoltageL1L2_V);
		x:=x+2;
		fb_Convert_Data(	word_In_1:= arrBuffer_Received[1,x], 
							word_In_2:= arrBuffer_Received[1,x+1], 
							e_ByteOrderIn:= e_ByteOrderConvert, 
							real_Output=> real_VoltageL2L3_V);
		x:=x+2;
		fb_Convert_Data(	word_In_1:= arrBuffer_Received[1,x], 
							word_In_2:= arrBuffer_Received[1,x+1], 
							e_ByteOrderIn:= e_ByteOrderConvert, 
							real_Output=> real_VoltageL3L1_V);
		x:=x+2;
		fb_Convert_Data(	word_In_1:= arrBuffer_Received[1,x], 
							word_In_2:= arrBuffer_Received[1,x+1], 
							e_ByteOrderIn:= e_ByteOrderConvert, 
							real_Output=> real_CurrentL1_A);
		x:=x+2;
		fb_Convert_Data(	word_In_1:= arrBuffer_Received[1,x], 
							word_In_2:= arrBuffer_Received[1,x+1], 
							e_ByteOrderIn:= e_ByteOrderConvert, 
							real_Output=> real_CurrentL2_A);
		x:=x+2;
		fb_Convert_Data(	word_In_1:= arrBuffer_Received[1,x], 
							word_In_2:= arrBuffer_Received[1,x+1], 
							e_ByteOrderIn:= e_ByteOrderConvert, 
							real_Output=> real_CurrentL3_A);		
		x:=24;
		fb_Convert_Data(	word_In_1:= arrBuffer_Received[1,x], 
							word_In_2:= arrBuffer_Received[1,x+1], 
							e_ByteOrderIn:= e_ByteOrderConvert, 
							real_Output=> real_RealPowerL1_kW);
							real_RealPowerL1_kW := real_RealPowerL1_kW/1000;
		x:=x+2;		
		fb_Convert_Data(	word_In_1:= arrBuffer_Received[1,x], 
							word_In_2:= arrBuffer_Received[1,x+1], 
							e_ByteOrderIn:= e_ByteOrderConvert, 
							real_Output=> real_RealPowerL2_kW);		
							real_RealPowerL2_kW := real_RealPowerL2_kW/1000;
		x:=x+2;		
		fb_Convert_Data(	word_In_1:= arrBuffer_Received[1,x], 
							word_In_2:= arrBuffer_Received[1,x+1], 
							e_ByteOrderIn:= e_ByteOrderConvert, 
							real_Output=> real_RealPowerL3_kW);
							real_RealPowerL3_kW := real_RealPowerL3_kW/1000;								
		x:=54;		
		fb_Convert_Data(	word_In_1:= arrBuffer_Received[1,x], 
							word_In_2:= arrBuffer_Received[1,x+1], 
							e_ByteOrderIn:= e_ByteOrderConvert, 
							real_Output=> real_Frequency_Hz);									
		x:=62;		
		fb_Convert_Data(	word_In_1:= arrBuffer_Received[1,x], 
							word_In_2:= arrBuffer_Received[1,x+1], 
							e_ByteOrderIn:= e_ByteOrderConvert, 
							real_Output=> real_ApparentPower_kVA);
							real_ApparentPower_kVA := real_ApparentPower_kVA/1000;									
		x:=x+2;	
		fb_Convert_Data(	word_In_1:= arrBuffer_Received[1,x], 
							word_In_2:= arrBuffer_Received[1,x+1], 
							e_ByteOrderIn:= e_ByteOrderConvert, 
							real_Output=> real_RealPower_kW);	
							real_RealPower_kW := real_RealPower_kW/1000;
		x:=x+2;	
		fb_Convert_Data(	word_In_1:= arrBuffer_Received[1,x], 
							word_In_2:= arrBuffer_Received[1,x+1], 
							e_ByteOrderIn:= e_ByteOrderConvert, 
							real_Output=> real_ReactivePower_kVAr);	
							real_ReactivePower_kVAr := real_ReactivePower_kVAr/1000;
		//2nd Poll
		x:=0;	
		fb_Convert_Data(	word_In_1:= arrBuffer_Received[2,x], 
							word_In_2:= arrBuffer_Received[2,x+1], 
							e_ByteOrderIn:= e_ByteOrderConvert, 
							real_Output=> real_EnergyTotal_Import_T1_kWh);		
							real_EnergyTotal_Import_T1_kWh := real_EnergyTotal_Import_T1_kWh/1000;
		x:=x+2;	
		fb_Convert_Data(	word_In_1:= arrBuffer_Received[2,x], 
							word_In_2:= arrBuffer_Received[2,x+1], 
							e_ByteOrderIn:= e_ByteOrderConvert, 
							real_Output=> real_EnergyTotal_Import_T2_kWh);		
							real_EnergyTotal_Import_T2_kWh := real_EnergyTotal_Import_T2_kWh/1000;
		x:=x+2;	
		fb_Convert_Data(	word_In_1:= arrBuffer_Received[2,x], 
							word_In_2:= arrBuffer_Received[2,x+1], 
							e_ByteOrderIn:= e_ByteOrderConvert, 
							real_Output=> real_EnergyTotal_Export_T1_kWh);	
							real_EnergyTotal_Export_T1_kWh := real_EnergyTotal_Export_T1_kWh/1000;	
		x:=x+2;	
		fb_Convert_Data(	word_In_1:= arrBuffer_Received[2,x], 
							word_In_2:= arrBuffer_Received[2,x+1], 
							e_ByteOrderIn:= e_ByteOrderConvert, 
							real_Output=> real_EnergyTotal_Export_T2_kWh);		
							real_EnergyTotal_Export_T2_kWh := real_EnergyTotal_Export_T2_kWh/1000;							

		
		// go to next state
		iStateModbusRead := iStateModbusRead+1;		
		
	31://Wait and go to start
		timer_Wait.IN := TRUE;
		
		IF timer_Wait.Q = TRUE THEN
			iStateModbusRead := 1;
			timer_Wait.IN :=FALSE;
		END_IF	

END_CASE

(* wait timer*)

timer_Wait(PT:=T#1S);


(*------------------------------------------------------------------Error and Warning----------------------------------------------------------------------------*)	
 
timer_Connection_ok			(In:=int_Data_Received<>int_Data_Received_old,PT:=T#10S);
timer_Connection_ok_TOF		(In:=NOT(int_Data_Received<>int_Data_Received_old) AND int_Data_Received>3 ,PT:=T#20S);
int_Data_Received_old:=int_Data_Received;
m_PollSuccessful:=NOT timer_Connection_ok.Q AND timer_Connection_ok_TOF.Q ;

(*------------------------------------------------------------------------------------------Modbus TCP Functions---------------------------------------------------------------------------------------------*)

fbMBRead_FC3(	sIPAddr:= str_IPAdress, 
				nTCPPort:= 502,
				cbLength:= SIZEOF(arrBuffer_FC3), 
				pDestAddr:= ADR(arrBuffer_FC3), 
				tTimeout:= T#10S,
				nErrId => udint_Error_ID);

FPError_FC_3(CLK:= fbMBRead_FC3.bError, Q=> );		

(*------------------------------------------------------------------------------------------State Machine Error---------------------------------------------------------------------------------------------*)	

CASE iStateModbusError OF
	
	300://Error
		timer_Wait.IN :=TRUE;
		timer_Delay.IN := FALSE;
		fbMBRead_FC3.bExecute := FALSE;
		m_MBTCPError := TRUE; 		
		m_Poll_ok:=FALSE;
		int_Data_Received:=0;
		
				//Restart from new with the Read out part after an Error
		IF timer_Wait.Q = TRUE THEN
			iStateModbusRead := 0;	
			iStateModbusError := 0;
			timer_Wait.IN :=FALSE;
			timer_Timeout.IN := FALSE;
		END_IF		
							
END_CASE

END_FUNCTION_BLOCK

// ---- FBs/prg_ReadDeviceName.TcPOU
PROGRAM prg_ReadDeviceName
VAR CONSTANT
	cNetId			: T_AmsNetID := '';				// local
END_VAR
VAR_INPUT
	bStart			: BOOL := TRUE;       			// flag to trigger (re)start of statemachine
END_VAR
VAR
	eState			: E_State := E_State.Init;
	hrGetValue		: HRESULT;	

	sDeviceName		: STRING(39);


	fbDiagRegister	: FB_IPCDiag_Register := (sNetId:=cNetId);
	fbDiagRead		: FB_IPCDiag_ReadParameter := (sNetId:=cNetId);
	nKeyIdx			: USINT := 1;
	aParameterKeys	: ARRAY[1..1] OF E_IPCDiag_ParameterKey := [	E_IPCDiag_ParameterKey.IPCDeviceName];
	ton_wait: Ton;
END_VAR

CASE eState OF
E_State.Init:
	IF NOT fbDiagRegister.bBusy THEN
		fbDiagRegister(bExecute:=TRUE); // need to be executed once
	ELSE
		fbDiagRegister(bExecute:=FALSE);
	END_IF
	IF NOT fbDiagRegister.bBusy THEN
		IF fbDiagRegister.bError THEN
			eState := E_State.Error;
		ELSE
			eState := E_State.Idle;
		END_IF
	END_IF

E_State.Idle:	
	ton_wait.IN := TRUE;
	IF ton_wait.Q THEN 
	    bStart := TRUE;	
		ton_wait.IN := FALSE;
	END_IF    
	IF bStart THEN
        bStart := FALSE;
        eState := E_State.ReadOnce;
    END_IF
	
E_State.ReadOnce: // reads every parameter once
	IF NOT fbDiagRead.bBusy THEN
		fbDiagRead(bExecute:= TRUE, eParameterKey:=aParameterKeys[nKeyIdx], fbRegister:=fbDiagRegister);	
	ELSE
		fbDiagRead(bExecute:= FALSE, fbRegister:=fbDiagRegister);
	END_IF
	IF NOT fbDiagRead.bBusy THEN
		IF fbDiagRead.bError OR FALSE THEN
			eState := E_State.Error;
		ELSE // get value
			IF aParameterKeys[nKeyIdx] = E_IPCDiag_ParameterKey.IPCDeviceName THEN
				hrGetValue := fbDiagRead.GetParameter(pBuffer:=ADR(sDeviceName), nBufferSize:=SIZEOF(sDeviceName));
			END_IF
				
			IF SUCCEEDED(hrGetValue) THEN
				eState := E_State.Wait;
			ELSE
				eState := E_State.Error;
			END_IF
		END_IF
	END_IF	

	
E_State.Error:
	(* implementation of error logging and error handling *)
	(* hint: An error could also occur if a parameter is not supported by chosen hardware or image. 
	E.g. not all IPCs offer a CPU temperature measurement. *)
	ton_wait.IN := TRUE;
	IF ton_wait.Q THEN 
		eState := E_State.Init;
		ton_wait.IN := FALSE;
	END_IF
	
E_State.Wait:	// wait for new trigger
	IF bStart THEN
		eState := E_State.Init;
	END_IF
	
END_CASE
ton_wait(PT := T#2S);

END_PROGRAM

// ---- POUs/prgCalc.TcPOU
PROGRAM prgCalc
VAR
	fbQ56Counter	: FB_EnergyCounter;
	lrPowerQ56		: LREAL;						//{#lynus.ag#()}
END_VAR
VAR PERSISTENT
	lrCounterQ56	: LREAL;						//{#lynus.ag#()}
	lrCO2Enphase	: LREAL;						//{#lynus.ag#()}
	lrCO2PV			: LREAL;						//{#lynus.ag#()}
END_VAR

// calc Output 5 & 6, 230V 16A, Schuko
// choose one of the two calc-options

// 1 -- if prgPV is in use
// lrPowerQ56 := (prgEM.lrPowerEM1 + prgBattery.lrPowerBatt + prgPV.lrPowerPV) - (prgEM.lrPowerEM2 + prgEM.lrPowerEM3 + prgEM.lrPowerEM4 + prgCS.lrPowerCS);
lrPowerQ56 := LIMIT(0,(prgEM.lrPowerEM1+ prgPV.lrPowerPV) - (prgEM.lrPowerEM2 + prgEM.lrPowerEM3 + prgEM.lrPowerEM4 + prgCS.lrPowerCS),10);

// 2 -- if prgEnphase is in use
// lrPowerQ56 := (prgEM.lrPowerEM1 + prgBattery.lrPowerBatt + prgEnphase.lrPowerPV) - (prgEM.lrPowerEM2 + prgEM.lrPowerEM3 + prgEM.lrPowerEM4 + prgCS.lrPowerCS);

fbQ56Counter(
	byActiveTariff:= 1, 
	lrPowerInput:= lrPowerQ56, 
	lrTotalCounterEnergy_Consumption=> , 
	lrTotalCounterEnergy_Production=> , 
	lrCounterEnergyT1_Consumption=> , 
	lrCounterEnergyT2_Consumption=> , 
	lrCounterEnergyT1_Production=> , 
	lrCounterEnergyT2_Production=> );
	
IF fbQ56Counter.lrTotalCounterEnergy_Consumption > lrCounterQ56 THEN  	
	lrCounterQ56 := fbQ56Counter.lrTotalCounterEnergy_Consumption;
END_IF

// calc saved CO2
// lrCO2Enphase := prgEnphase.lrCounterPV * 0.428;
lrCO2PV := prgPV.lrCounterPV * 0.428;

END_PROGRAM

// ---- POUs/prgEM.TcPOU
PROGRAM prgEM
VAR
	fbKBusState		: FB_K_Bus_State;
	fbEM1			: FB_EM_Beckhoff_KL3403;
	fbEM1Counter	: FB_EnergyCounter;
	fbEM2			: FB_EM_Beckhoff_KL3403;
	fbEM2Counter	: FB_EnergyCounter;
	fbEM3			: FB_EM_Beckhoff_KL3403;
	fbEM3Counter	: FB_EnergyCounter;
	fbEM4			: FB_EM_Beckhoff_KL3403;
	fbEM4Counter	: FB_EnergyCounter;
	fbEM5			: FB_EM_Beckhoff_KL3403;		// only EIOPL020004		Main supply
													// only EIOPL020013		extra measurement
	fbEM5Counter	: FB_EnergyCounter;
	fbEM6			: FB_EM_Beckhoff_KL3403;		// only EIOPL020004		Crane
													// only EIOPL020013		extra measurement
	fbEM6Counter	: FB_EnergyCounter;
	fbEM7			: FB_EM_Beckhoff_KL3403;		// only EIOPL020013		extra measurement
	fbEM7Counter	: FB_EnergyCounter;
		
	lrPowerEM1		: LREAL;							//{#lynus.ag#()}
	lrPowerEM2		: LREAL;							//{#lynus.ag#()}
	lrPowerEM3		: LREAL;							//{#lynus.ag#()}
	lrPowerEM4		: LREAL;							//{#lynus.ag#()}
	lrPowerEM5		: LREAL;							//{#lynus.ag#()}
	lrPowerEM6		: LREAL;							//{#lynus.ag#()}
	lrPowerEM7		: LREAL;							//{#lynus.ag#()}
	lr_InputVoltage_L1N		: LREAL;					//{#lynus.ag#()}
	lr_InputVoltage_L2N		: LREAL;					//{#lynus.ag#()}
	lr_InputVoltage_L3N		: LREAL;					//{#lynus.ag#()}
	lr_InputVoltage_L1L2	: LREAL;					//{#lynus.ag#()}
	lr_InputVoltage_L2L3	: LREAL;					//{#lynus.ag#()}
	lr_InputVoltage_L3L1	: LREAL;					//{#lynus.ag#()}
	lr_Power_EM1_L1	: LREAL;							//{#lynus.ag#()}
	lr_Power_EM1_L2	: LREAL;							//{#lynus.ag#()}
	lr_Power_EM1_L3	: LREAL;							//{#lynus.ag#()}
	lr_Power_EM2_L1	: LREAL;							//{#lynus.ag#()}
	lr_Power_EM2_L2	: LREAL;							//{#lynus.ag#()}
	lr_Power_EM2_L3	: LREAL;							//{#lynus.ag#()}
	lr_Power_EM3_L1	: LREAL;							//{#lynus.ag#()}
	lr_Power_EM3_L2	: LREAL;							//{#lynus.ag#()}
	lr_Power_EM3_L3	: LREAL;							//{#lynus.ag#()}
	lr_Power_EM4_L1	: LREAL;							//{#lynus.ag#()}
	lr_Power_EM4_L2	: LREAL;							//{#lynus.ag#()}
	lr_Power_EM4_L3	: LREAL;							//{#lynus.ag#()}
	lr_Power_EM5_L1	: LREAL;							//{#lynus.ag#()}
	lr_Power_EM5_L2	: LREAL;							//{#lynus.ag#()}
	lr_Power_EM5_L3	: LREAL;							//{#lynus.ag#()}
	lr_Power_EM6_L1	: LREAL;							//{#lynus.ag#()}
	lr_Power_EM6_L2	: LREAL;							//{#lynus.ag#()}
	lr_Power_EM6_L3	: LREAL;							//{#lynus.ag#()}
	lr_Power_EM7_L1	: LREAL;							//{#lynus.ag#()}
	lr_Power_EM7_L2	: LREAL;							//{#lynus.ag#()}
	lr_Power_EM7_L3	: LREAL;							//{#lynus.ag#()}
	lr_ReactivePower_EM1_Total	: LREAL;				//{#lynus.ag#()}
	lr_ApparentPower_EM1_Total	: LREAL;				//{#lynus.ag#()}
	lr_ReactivePower_EM2_Total	: LREAL;				//{#lynus.ag#()}
	lr_ApparentPower_EM2_Total	: LREAL;				//{#lynus.ag#()}
	lr_ReactivePower_EM3_Total	: LREAL;				//{#lynus.ag#()}
	lr_ApparentPower_EM3_Total	: LREAL;				//{#lynus.ag#()}
	lr_ReactivePower_EM4_Total	: LREAL;				//{#lynus.ag#()}
	lr_ApparentPower_EM4_Total	: LREAL;				//{#lynus.ag#()}
	lr_ReactivePower_EM5_Total	: LREAL;				//{#lynus.ag#()}
	lr_ApparentPower_EM5_Total	: LREAL;				//{#lynus.ag#()}
	lr_ReactivePower_EM6_Total	: LREAL;				//{#lynus.ag#()}
	lr_ApparentPower_EM6_Total	: LREAL;				//{#lynus.ag#()}
	lr_ReactivePower_EM7_Total	: LREAL;				//{#lynus.ag#()}
	lr_ApparentPower_EM7_Total	: LREAL;				//{#lynus.ag#()}
	lr_Frequency_EM1	: LREAL;						//{#lynus.ag#()}
	lr_Frequency_EM2	: LREAL;						//{#lynus.ag#()}
	lr_Frequency_EM3	: LREAL;						//{#lynus.ag#()}
	lr_Frequency_EM4	: LREAL;						//{#lynus.ag#()}
	lr_Frequency_EM5	: LREAL;						//{#lynus.ag#()}
	lr_Frequency_EM6	: LREAL;						//{#lynus.ag#()}
	lr_Frequency_EM7	: LREAL;						//{#lynus.ag#()}
	r_PowerFactor_EM1_L1: REAL;						//{#lynus.ag#()}
	r_PowerFactor_EM1_L2: REAL;						//{#lynus.ag#()}
	r_PowerFactor_EM1_L3: REAL;						//{#lynus.ag#()}
	r_PowerFactor_EM2_L1: REAL;						//{#lynus.ag#()}
	r_PowerFactor_EM2_L2: REAL;						//{#lynus.ag#()}
	r_PowerFactor_EM2_L3: REAL;						//{#lynus.ag#()}
	r_PowerFactor_EM3_L1: REAL;						//{#lynus.ag#()}
	r_PowerFactor_EM3_L2: REAL;						//{#lynus.ag#()}
	r_PowerFactor_EM3_L3: REAL;						//{#lynus.ag#()}
	r_PowerFactor_EM4_L1: REAL;						//{#lynus.ag#()}
	r_PowerFactor_EM4_L2: REAL;						//{#lynus.ag#()}
	r_PowerFactor_EM4_L3: REAL;						//{#lynus.ag#()}
	r_PowerFactor_EM5_L1: REAL;						//{#lynus.ag#()}
	r_PowerFactor_EM5_L2: REAL;						//{#lynus.ag#()}
	r_PowerFactor_EM5_L3: REAL;						//{#lynus.ag#()}
	r_PowerFactor_EM6_L1: REAL;						//{#lynus.ag#()}
	r_PowerFactor_EM6_L2: REAL;						//{#lynus.ag#()}
	r_PowerFactor_EM6_L3: REAL;						//{#lynus.ag#()}
	r_PowerFactor_EM7_L1: REAL;						//{#lynus.ag#()}
	r_PowerFactor_EM7_L2: REAL;						//{#lynus.ag#()}
	r_PowerFactor_EM7_L3: REAL;						//{#lynus.ag#()}
	
	
END_VAR
VAR_INPUT
	uiCurrentTransformerRatioL1	:UINT;
	uiCurrentTransformerRatioL2	:UINT;
	uiCurrentTransformerRatioL3	:UINT;	
END_VAR
VAR PERSISTENT
	lrCounterEM1	: LREAL;						//{#lynus.ag#()}
	lrCounterEM2	: LREAL;						//{#lynus.ag#()}
	lrCounterEM3	: LREAL;						//{#lynus.ag#()}
	lrCounterEM4	: LREAL;						//{#lynus.ag#()}
	lrCounterEM5	: LREAL;						//{#lynus.ag#()}
	lrCounterEM6	: LREAL;						//{#lynus.ag#()}
	lrCounterEM7	: LREAL;						//{#lynus.ag#()}
END_VAR

fbKBusState(	uiKBusState_OUT=> , 
				b_Kbus_notOk=> , 
				word_ErrorCount=> );


fbEM1(
	bEnable:= TRUE, 
	bChannel1Invers:= FALSE,
	bChannel2Invers:= FALSE,
	bChannel3Invers:= FALSE,
	uiCurrentTransformerRatioL1:= uiCurrentTransformerRatioL1, 
	uiCurrentTransformerRatioL2:= uiCurrentTransformerRatioL2, 
	uiCurrentTransformerRatioL3:= uiCurrentTransformerRatioL3, 
	uiKBusState_IN:= fbKBusState.uiKBusState_OUT, 
	stDataEMPower=> , 
	stDataEMCounter=> , 
	stDataEMPowerRealTime=> , 
	stDataEMCounterRealTime=> , 
	diNrOfEM_OUT=> );

lrPowerEM1 := fbEM1.stDataEMPower.lrPowerTotal;	
lr_InputVoltage_L1N := fbEM1.stDataEMPower.lrVoltageL1N;
lr_InputVoltage_L2N := fbEM1.stDataEMPower.lrVoltageL2N;
lr_InputVoltage_L3N := fbEM1.stDataEMPower.lrVoltageL3N;
lr_InputVoltage_L1L2 := fbEM1.stDataEMPower.lrVoltageL1L2;
lr_InputVoltage_L2L3 := fbEM1.stDataEMPower.lrVoltageL2L3;
lr_InputVoltage_L3L1 := fbEM1.stDataEMPower.lrVoltageL3L1;

fbEM1Counter(
	byActiveTariff:= 1, 
	lrPowerInput:= lrPowerEM1, 
	lrTotalCounterEnergy_Consumption=> , 
	lrTotalCounterEnergy_Production=> , 
	lrCounterEnergyT1_Consumption=> , 
	lrCounterEnergyT2_Consumption=> , 
	lrCounterEnergyT1_Production=> , 
	lrCounterEnergyT2_Production=> );
	
IF fbEM1Counter.lrTotalCounterEnergy_Consumption > lrCounterEM1 THEN  	
	lrCounterEM1 := fbEM1Counter.lrTotalCounterEnergy_Consumption;
END_IF

// Output1, 3x400V 32A, CEE32

fbEM2(
	bEnable:= TRUE, 
	bChannel1Invers:= FALSE,
	bChannel2Invers:= FALSE,
	bChannel3Invers:= FALSE,
	uiCurrentTransformerRatioL1:= 35, 
	uiCurrentTransformerRatioL2:= 35, 
	uiCurrentTransformerRatioL3:= 35, 
	uiKBusState_IN:= fbKBusState.uiKBusState_OUT, 
	stDataEMPower=> , 
	stDataEMCounter=> , 
	stDataEMPowerRealTime=> , 
	stDataEMCounterRealTime=> , 
	diNrOfEM_OUT=> );

lrPowerEM2 := fbEM2.stDataEMPower.lrPowerTotal;	

fbEM2Counter(
	byActiveTariff:= 1, 
	lrPowerInput:= lrPowerEM2, 
	lrTotalCounterEnergy_Consumption=> , 
	lrTotalCounterEnergy_Production=> , 
	lrCounterEnergyT1_Consumption=> , 
	lrCounterEnergyT2_Consumption=> , 
	lrCounterEnergyT1_Production=> , 
	lrCounterEnergyT2_Production=> );
	
IF fbEM2Counter.lrTotalCounterEnergy_Consumption > lrCounterEM2 THEN  	
	lrCounterEM2 := fbEM2Counter.lrTotalCounterEnergy_Consumption;
END_IF


// Output2, 3x400V 32A, CEE32

fbEM3(
	bEnable:= TRUE, 
	bChannel1Invers:= FALSE,
	bChannel2Invers:= FALSE,
	bChannel3Invers:= FALSE,
	uiCurrentTransformerRatioL1:= 35, 
	uiCurrentTransformerRatioL2:= 35, 
	uiCurrentTransformerRatioL3:= 35, 
	uiKBusState_IN:= fbKBusState.uiKBusState_OUT, 
	stDataEMPower=> , 
	stDataEMCounter=> , 
	stDataEMPowerRealTime=> , 
	stDataEMCounterRealTime=> , 
	diNrOfEM_OUT=> );

lrPowerEM3 := fbEM3.stDataEMPower.lrPowerTotal;	

fbEM3Counter(
	byActiveTariff:= 1, 
	lrPowerInput:= lrPowerEM3, 
	lrTotalCounterEnergy_Consumption=> , 
	lrTotalCounterEnergy_Production=> , 
	lrCounterEnergyT1_Consumption=> , 
	lrCounterEnergyT2_Consumption=> , 
	lrCounterEnergyT1_Production=> , 
	lrCounterEnergyT2_Production=> );
	
IF fbEM3Counter.lrTotalCounterEnergy_Consumption > lrCounterEM3 THEN  	
	lrCounterEM3 := fbEM3Counter.lrTotalCounterEnergy_Consumption;
END_IF


// Output3, 3x400V 16A, CEE16

fbEM4(
	bEnable:= TRUE, 
	bChannel1Invers:= FALSE,
	bChannel2Invers:= FALSE,
	bChannel3Invers:= FALSE,
	uiCurrentTransformerRatioL1:= 35, 
	uiCurrentTransformerRatioL2:= 35, 
	uiCurrentTransformerRatioL3:= 35, 
	uiKBusState_IN:= fbKBusState.uiKBusState_OUT, 
	stDataEMPower=> , 
	stDataEMCounter=> , 
	stDataEMPowerRealTime=> , 
	stDataEMCounterRealTime=> , 
	diNrOfEM_OUT=> );

lrPowerEM4 := fbEM4.stDataEMPower.lrPowerTotal;	

fbEM4Counter(
	byActiveTariff:= 1, 
	lrPowerInput:= lrPowerEM4, 
	lrTotalCounterEnergy_Consumption=> , 
	lrTotalCounterEnergy_Production=> , 
	lrCounterEnergyT1_Consumption=> , 
	lrCounterEnergyT2_Consumption=> , 
	lrCounterEnergyT1_Production=> , 
	lrCounterEnergyT2_Production=> );
	
IF fbEM4Counter.lrTotalCounterEnergy_Consumption > lrCounterEM4 THEN  	
	lrCounterEM4 := fbEM4Counter.lrTotalCounterEnergy_Consumption;
END_IF


// only EIOPL02004

fbEM5(
	bEnable:= TRUE, 
	bChannel1Invers:= FALSE,
	bChannel2Invers:= FALSE,
	bChannel3Invers:= FALSE,
	uiCurrentTransformerRatioL1:= 400, 
	uiCurrentTransformerRatioL2:= 400, 
	uiCurrentTransformerRatioL3:= 400, 
	uiKBusState_IN:= fbKBusState.uiKBusState_OUT, 
	stDataEMPower=> , 
	stDataEMCounter=> , 
	stDataEMPowerRealTime=> , 
	stDataEMCounterRealTime=> , 
	diNrOfEM_OUT=> );
lrPowerEM5 := fbEM5.stDataEMPower.lrPowerTotal;	
	
fbEM5Counter(
	byActiveTariff:= 1, 
	lrPowerInput:= lrPowerEM5, 
	lrTotalCounterEnergy_Consumption=> , 
	lrTotalCounterEnergy_Production=> , 
	lrCounterEnergyT1_Consumption=> , 
	lrCounterEnergyT2_Consumption=> , 
	lrCounterEnergyT1_Production=> , 
	lrCounterEnergyT2_Production=> );
	
IF fbEM5Counter.lrTotalCounterEnergy_Consumption > lrCounterEM5 THEN  	
	lrCounterEM5 := fbEM5Counter.lrTotalCounterEnergy_Consumption;
END_IF

fbEM6(
	bEnable:= TRUE, 
	bChannel1Invers:= FALSE,
	bChannel2Invers:= FALSE,
	bChannel3Invers:= FALSE,
	uiCurrentTransformerRatioL1:= 400, 
	uiCurrentTransformerRatioL2:= 400, 
	uiCurrentTransformerRatioL3:= 400, 
	uiKBusState_IN:= fbKBusState.uiKBusState_OUT, 
	stDataEMPower=> , 
	stDataEMCounter=> , 
	stDataEMPowerRealTime=> , 
	stDataEMCounterRealTime=> , 
	diNrOfEM_OUT=> );
lrPowerEM6 := fbEM6.stDataEMPower.lrPowerTotal;	

fbEM6Counter(
	byActiveTariff:= 1, 
	lrPowerInput:= lrPowerEM6, 
	lrTotalCounterEnergy_Consumption=> , 
	lrTotalCounterEnergy_Production=> , 
	lrCounterEnergyT1_Consumption=> , 
	lrCounterEnergyT2_Consumption=> , 
	lrCounterEnergyT1_Production=> , 
	lrCounterEnergyT2_Production=> );
	
IF fbEM6Counter.lrTotalCounterEnergy_Consumption > lrCounterEM6 THEN  	
	lrCounterEM6 := fbEM6Counter.lrTotalCounterEnergy_Consumption;
END_IF

fbEM7(
	bEnable:= TRUE, 
	bChannel1Invers:= FALSE,
	bChannel2Invers:= FALSE,
	bChannel3Invers:= FALSE,
	uiCurrentTransformerRatioL1:= 400, 
	uiCurrentTransformerRatioL2:= 400, 
	uiCurrentTransformerRatioL3:= 400, 
	uiKBusState_IN:= fbKBusState.uiKBusState_OUT, 
	stDataEMPower=> , 
	stDataEMCounter=> , 
	stDataEMPowerRealTime=> , 
	stDataEMCounterRealTime=> , 
	diNrOfEM_OUT=> );
lrPowerEM7 := fbEM7.stDataEMPower.lrPowerTotal;	

fbEM6Counter(
	byActiveTariff:= 1, 
	lrPowerInput:= lrPowerEM7, 
	lrTotalCounterEnergy_Consumption=> , 
	lrTotalCounterEnergy_Production=> , 
	lrCounterEnergyT1_Consumption=> , 
	lrCounterEnergyT2_Consumption=> , 
	lrCounterEnergyT1_Production=> , 
	lrCounterEnergyT2_Production=> );
	
IF fbEM7Counter.lrTotalCounterEnergy_Consumption > lrCounterEM7 THEN  	
	lrCounterEM7 := fbEM7Counter.lrTotalCounterEnergy_Consumption;
END_IF

// additinal data sent to cloud
lr_Power_EM1_L1 			:=	fbEM1.stDataEMPowerRealTime.lrPowerL1;
lr_Power_EM1_L2 			:=	fbEM1.stDataEMPowerRealTime.lrPowerL2;
lr_Power_EM1_L3 			:=	fbEM1.stDataEMPowerRealTime.lrPowerL3;
lr_ReactivePower_EM1_Total	:= 	fbEM1.stDataEMPowerRealTime.lrReactivePowerTotal;
lr_ApparentPower_EM1_Total	:= 	fbEM1.stDataEMPowerRealTime.lrApparentPowerTotal;
lr_Frequency_EM1			:= 	fbEM1.stDataEMPowerRealTime.lrFrequency;
r_PowerFactor_EM1_L1		:=	fbEM1.fbKL3403.stDataL1.rPowerfactor;
r_PowerFactor_EM1_L2		:=	fbEM1.fbKL3403.stDataL2.rPowerfactor;
r_PowerFactor_EM1_L3		:=	fbEM1.fbKL3403.stDataL3.rPowerfactor;

lr_Power_EM2_L1 			:=	fbEM2.stDataEMPowerRealTime.lrPowerL1;
lr_Power_EM2_L2 			:=	fbEM2.stDataEMPowerRealTime.lrPowerL2;
lr_Power_EM2_L3 			:=	fbEM2.stDataEMPowerRealTime.lrPowerL3;
lr_ReactivePower_EM2_Total	:= 	fbEM2.stDataEMPowerRealTime.lrReactivePowerTotal;
lr_ApparentPower_EM2_Total	:= 	fbEM2.stDataEMPowerRealTime.lrApparentPowerTotal;
lr_Frequency_EM2			:= 	fbEM2.stDataEMPowerRealTime.lrFrequency;
r_PowerFactor_EM2_L1		:=	fbEM2.fbKL3403.stDataL1.rPowerfactor;
r_PowerFactor_EM2_L2		:=	fbEM2.fbKL3403.stDataL2.rPowerfactor;
r_PowerFactor_EM2_L3		:=	fbEM2.fbKL3403.stDataL3.rPowerfactor;

lr_Power_EM3_L1 			:=	fbEM3.stDataEMPowerRealTime.lrPowerL1;
lr_Power_EM3_L2 			:=	fbEM3.stDataEMPowerRealTime.lrPowerL2;
lr_Power_EM3_L3 			:=	fbEM3.stDataEMPowerRealTime.lrPowerL3;
lr_ReactivePower_EM3_Total	:= 	fbEM3.stDataEMPowerRealTime.lrReactivePowerTotal;
lr_ApparentPower_EM3_Total	:= 	fbEM3.stDataEMPowerRealTime.lrApparentPowerTotal;
lr_Frequency_EM3			:= 	fbEM3.stDataEMPowerRealTime.lrFrequency;
r_PowerFactor_EM3_L1		:=	fbEM3.fbKL3403.stDataL1.rPowerfactor;
r_PowerFactor_EM3_L2		:=	fbEM3.fbKL3403.stDataL2.rPowerfactor;
r_PowerFactor_EM3_L3		:=	fbEM3.fbKL3403.stDataL3.rPowerfactor;

lr_Power_EM4_L1 			:=	fbEM4.stDataEMPowerRealTime.lrPowerL1;
lr_Power_EM4_L2 			:=	fbEM4.stDataEMPowerRealTime.lrPowerL2;
lr_Power_EM4_L3 			:=	fbEM4.stDataEMPowerRealTime.lrPowerL3;
lr_ReactivePower_EM4_Total	:= 	fbEM4.stDataEMPowerRealTime.lrReactivePowerTotal;
lr_ApparentPower_EM4_Total	:= 	fbEM4.stDataEMPowerRealTime.lrApparentPowerTotal;
lr_Frequency_EM4			:= 	fbEM4.stDataEMPowerRealTime.lrFrequency;
r_PowerFactor_EM4_L1		:=	fbEM4.fbKL3403.stDataL1.rPowerfactor;
r_PowerFactor_EM4_L2		:=	fbEM4.fbKL3403.stDataL2.rPowerfactor;
r_PowerFactor_EM4_L3		:=	fbEM4.fbKL3403.stDataL3.rPowerfactor;

lr_Power_EM5_L1 			:=	fbEM5.stDataEMPowerRealTime.lrPowerL1;
lr_Power_EM5_L2 			:=	fbEM5.stDataEMPowerRealTime.lrPowerL2;
lr_Power_EM5_L3 			:=	fbEM5.stDataEMPowerRealTime.lrPowerL3;
lr_ReactivePower_EM5_Total	:= 	fbEM5.stDataEMPowerRealTime.lrReactivePowerTotal;
lr_ApparentPower_EM5_Total	:= 	fbEM5.stDataEMPowerRealTime.lrApparentPowerTotal;
lr_Frequency_EM5			:= 	fbEM5.stDataEMPowerRealTime.lrFrequency;
r_PowerFactor_EM5_L1		:=	fbEM5.fbKL3403.stDataL1.rPowerfactor;
r_PowerFactor_EM5_L2		:=	fbEM5.fbKL3403.stDataL2.rPowerfactor;
r_PowerFactor_EM5_L3		:=	fbEM5.fbKL3403.stDataL3.rPowerfactor;

lr_Power_EM6_L1 			:=	fbEM6.stDataEMPowerRealTime.lrPowerL1;
lr_Power_EM6_L2 			:=	fbEM6.stDataEMPowerRealTime.lrPowerL2;
lr_Power_EM6_L3 			:=	fbEM6.stDataEMPowerRealTime.lrPowerL3;
lr_ReactivePower_EM6_Total	:= 	fbEM6.stDataEMPowerRealTime.lrReactivePowerTotal;
lr_ApparentPower_EM6_Total	:= 	fbEM6.stDataEMPowerRealTime.lrApparentPowerTotal;
lr_Frequency_EM6			:= 	fbEM6.stDataEMPowerRealTime.lrFrequency;
r_PowerFactor_EM6_L1		:=	fbEM6.fbKL3403.stDataL1.rPowerfactor;
r_PowerFactor_EM6_L2		:=	fbEM6.fbKL3403.stDataL2.rPowerfactor;
r_PowerFactor_EM6_L3		:=	fbEM6.fbKL3403.stDataL3.rPowerfactor;

lr_Power_EM7_L1 			:=	fbEM7.stDataEMPowerRealTime.lrPowerL1;
lr_Power_EM7_L2 			:=	fbEM7.stDataEMPowerRealTime.lrPowerL2;
lr_Power_EM7_L3 			:=	fbEM7.stDataEMPowerRealTime.lrPowerL3;
lr_ReactivePower_EM7_Total	:= 	fbEM7.stDataEMPowerRealTime.lrReactivePowerTotal;
lr_ApparentPower_EM7_Total	:= 	fbEM7.stDataEMPowerRealTime.lrApparentPowerTotal;
lr_Frequency_EM7			:= 	fbEM7.stDataEMPowerRealTime.lrFrequency;
r_PowerFactor_EM7_L1		:=	fbEM7.fbKL3403.stDataL1.rPowerfactor;
r_PowerFactor_EM7_L2		:=	fbEM7.fbKL3403.stDataL2.rPowerfactor;
r_PowerFactor_EM7_L3		:=	fbEM7.fbKL3403.stDataL3.rPowerfactor;

END_PROGRAM

// ---- POUs/prgPV.TcPOU
PROGRAM prgPV
VAR
	fbPV						: FB_Hoymiles_DTU_ProS_PV_Inverter_inclWrite;
//	fbPV						: FB_Hoymiles_DTU_ProS_PV_Inverter;
	fbEnphase					: FB_Enphase;
	fbPVCounter					: FB_EnergyCounter;
	lrPowerPVEnphase_W			: LREAL;
	lrPowerPV					: LREAL;						//{#lynus.ag#()}
	byErrorWarningPV			: BYTE;							//{#lynus.ag#()}
	fbEM						: FB_EM_Beckhoff_KL3403;
	byte_Setpoint				: BYTE := 100;
END_VAR
VAR_INPUT
	m_Hoymiles_DTU_ProS_PV_Inverter		: BOOL;
	m_Enphase							: BOOL;
	m_KL3403							: BOOL;	
END_VAR
VAR PERSISTENT
	lrCounterPV					: LREAL;						//{#lynus.ag#()}
	bEnable						: BOOL;
	str_IP						: STRING(15);
END_VAR

// To-Do:
// adopt FB Declaration, change to correct FB
// adopt FB Definition, change to correct in/out Vars
// correct lrPowerPV definition
// correct lrCounterPV definition
// correct byErrorWarningPV definition


// PV config for external Inverter

IF m_Hoymiles_DTU_ProS_PV_Inverter = TRUE THEN
	fbPV(
		bEnable:= bEnable, 
		sIPAdress:= str_IP, 
		byUnitID_Inverter:= 101, 
		byte_Setpoint:= byte_Setpoint, 
		DataHoymiles_DTU_Pro_Total=> , 
		arrDataHoymiles_DTU_Pro=> , 
		stDataEMPower_PV=> , 
		stDataEMCounter_PV=> , 
		diNrOfEM_OUT_PV=> );

	// operation state of the inverter is unclear if that is ok, no documentation from Hoymiles
	
	lrPowerPV := fbPV.DataHoymiles_DTU_Pro_Total.lrPowerAcInverter;
	byErrorWarningPV := fbPV.stDataEMPower_PV.byErrorWarning;
	
	IF fbPV.stDataEMCounter_PV.lrCounterEnergyT1_Production > lrCounterPV THEN  	
		lrCounterPV := fbPV.stDataEMCounter_PV.lrCounterEnergyT1_Production;
	END_IF

END_IF


// PV config for Enphase Gateway			--> only PowerLink #2
IF m_Enphase THEN
	
	fbEnphase(
		bStart:= TRUE, 
		tDelayRequest:= T#3S, 
//		sHostname:= '192.168.1.231', 		EIOPL020003 / Stuttgart
		sHostname:= '192.168.1.30',  
		bValidResult=> , 
		bBusy=> , 
		bError=> , 
		bDone=> , 
		hrErrorCode=> ,
		lrpowerprod => lrPowerPVEnphase_W );
		
	// re-calc Power to kW
	lrPowerPV := lrPowerPVEnphase_W / 1000;
	
	fbPVCounter(
		byActiveTariff:= 1, 
		lrPowerInput:= lrPowerPV, 
		lrTotalCounterEnergy_Consumption=> , 
		lrTotalCounterEnergy_Production=> , 
		lrCounterEnergyT1_Consumption=> , 
		lrCounterEnergyT2_Consumption=> , 
		lrCounterEnergyT1_Production=> , 
		lrCounterEnergyT2_Production=> );
		
	IF fbPVCounter.lrTotalCounterEnergy_Consumption > lrCounterPV THEN  	
		lrCounterPV := fbPVCounter.lrTotalCounterEnergy_Consumption;
	END_IF
END_IF

IF m_KL3403 THEN 
	fbEM(
		bEnable:= TRUE, 
		bChannel1Invers:= FALSE,
		bChannel2Invers:= FALSE,
		bChannel3Invers:= FALSE,
		uiCurrentTransformerRatioL1:= 35, 
		uiCurrentTransformerRatioL2:= 35, 
		uiCurrentTransformerRatioL3:= 35, 
		uiKBusState_IN:= prgEM.fbKBusState.uiKBusState_OUT, 
		stDataEMPower=> , 
		stDataEMCounter=> , 
		stDataEMPowerRealTime=> , 
		stDataEMCounterRealTime=> , 
		diNrOfEM_OUT=> );
		
	lrPowerPV := fbEM.stDataEMPower.lrPowerProduction;
	
	fbPVCounter(
		byActiveTariff:= 1, 
		lrPowerInput:= lrPowerPV, 
		lrTotalCounterEnergy_Consumption=> , 
		lrTotalCounterEnergy_Production=> , 
		lrCounterEnergyT1_Consumption=> , 
		lrCounterEnergyT2_Consumption=> , 
		lrCounterEnergyT1_Production=> , 
		lrCounterEnergyT2_Production=> );
		
	IF fbPVCounter.lrTotalCounterEnergy_Consumption > lrCounterPV THEN  	
		lrCounterPV := fbPVCounter.lrTotalCounterEnergy_Consumption;
	END_IF
	
END_IF

END_PROGRAM

// ---- POUs/prgCS.TcPOU
PROGRAM prgCS
VAR
	fbCS						: FB_EM24_DIN; 
	fbCS_2						: FB_PAC2200; 
	fbCSCounter					: FB_EnergyCounter;
	lrPowerCS					: LREAL;						//{#lynus.ag#()}
	// udintErrorWarningCS			: UDINT;
	FB_MB_Test :FB_ModBus_100Registers_FC3_inclID;
	
	fbLIBREO_1					: FB_ECS_LIBREO;
	bEnable_LIBREO_1			: BOOL;
	bCarConnected_LIBREO_1				: BOOL;						//{#lynus.ag#()}
	bCarCharging_LIBREO_1				: BOOL;						//{#lynus.ag#()}
	lrTotalPower_LIBREO_1				: LREAL;					//{#lynus.ag#()}
	uiChrgCurr_LIBREO_1					: UINT;						//{#lynus.ag#()}
	uiExtChrgCurr_LIBREO_1				: UINT;						//{#lynus.ag#()}
	bCarConnLED_LIBREO_1				: UINT;						//{#lynus.ag#()}
END_VAR
VAR_INPUT
	m_EM24_DIN					: BOOL;
	m_PAC2200					: BOOL;
END_VAR
VAR PERSISTENT
	lrCounterCS					: LREAL;						//{#lynus.ag#()}
	lrCounterCSeIO				: LREAL;						//{#lynus.ag#()}
END_VAR

// To-Do:
// adopt FB Declaration, change to new FB for ENERGYMID
// adopt FB Definition, change to correct in/out Vars for ENERGYMID
// correct lrPowerCS definition
// correct lrCounterCS definition
// correct byErrorWarningCS definition

IF 	m_PAC2200 THEN 
	fbCS_2(
		m_Enable:= TRUE, 
		str_IPAdress:=  '192.168.1.20',   
		real_RealPower_kW=> , 
		real_RealPowerL1_kW=> , 
		real_RealPowerL2_kW=> , 
		real_RealPowerL3_kW=> , 
		real_ReactivePower_kVAr=> , 
		real_ApparentPower_kVA=> , 
		real_Frequency_Hz=> , 
		real_VoltageL1N_V=> , 
		real_VoltageL2N_V=> , 
		real_VoltageL3N_V=> , 
		real_VoltageL1L2_V=> , 
		real_VoltageL2L3_V=> , 
		real_VoltageL3L1_V=> , 
		real_CurrentL1_A=> , 
		real_CurrentL2_A=> , 
		real_CurrentL3_A=> , 
		real_EnergyTotal_Import_T1_kWh=> , 
		real_EnergyTotal_Import_T2_kWh=> , 
		real_EnergyTotal_Export_T1_kWh=> , 
		real_EnergyTotal_Export_T2_kWh=> , 
		m_PollSuccessful=> , 
		udint_Error_ID=> );
		
	lrPowerCS := fbCS_2.real_RealPower_kW;
	// uErrorWarningCS := fbCS.udint_Error_ID;
	
	// MID conform Counter, read from Energymeter
	IF fbCS_2.real_EnergyTotal_Import_T1_kWh > lrCounterCS THEN  	
		lrCounterCS := fbCS_2.real_EnergyTotal_Import_T1_kWh;
	END_IF
	
	// internal Counter, for comparing purpose
	fbCSCounter(
		byActiveTariff:= 1, 
		lrPowerInput:= lrPowerCS, 
		lrTotalCounterEnergy_Consumption=> , 
		lrTotalCounterEnergy_Production=> , 
		lrCounterEnergyT1_Consumption=> , 
		lrCounterEnergyT2_Consumption=> , 
		lrCounterEnergyT1_Production=> , 
		lrCounterEnergyT2_Production=> );
		
